(* IEC 61131-3 sources: Yaha/Documentation/Infomaterial/OSCAT/pcworx_basic_333/module_export (part 7) *)

(* ---- BIT_LOAD_DW.ST ---- *)
(*@PROPERTIES_EX@
TYPE: POU
LOCALE: 0
IEC_LANGUAGE: ST
PLC_TYPE: independent
PROC_TYPE: independent
GROUP: LOGIC.GATE_LOGIC
*)
(*@KEY@:DESCRIPTION*)
version 1.1	16. mar 2008
programmer 	hugo
tested by	tobias

this function loads a bit into a DWord at position pos.
(*@KEY@:END_DESCRIPTION*)
FUNCTION BIT_LOAD_DW:DWORD

(*Group:Default*)

VAR_INPUT
	IN :	DWORD;
	VAL :	BOOL;
	POS :	INT;
END_VAR

(*@KEY@: WORKSHEET
NAME: BIT_LOAD_DW
IEC_LANGUAGE: ST
*)
IF val THEN
	BIT_LOAD_DW := in OR SHL(DWORD#1,pos);
ELSE
	BIT_LOAD_DW := in AND (NOT SHL(DWORD#1,pos));
END_IF;

(* revision history
hm	29. feb 2008	rev 1.0
	original version

hm	16. mar 2008	rev 1.1
	change input bit to val for compatibility reasons
*)
(*@KEY@: END_WORKSHEET *)
END_FUNCTION

(* ---- BIT_LOAD_DW2.ST ---- *)
(*@PROPERTIES_EX@
TYPE: POU
LOCALE: 0
IEC_LANGUAGE: ST
PLC_TYPE: independent
PROC_TYPE: independent
GROUP: LOGIC.GATE_LOGIC
*)
(*@KEY@:DESCRIPTION*)
version 1.0 18. oct. 2008
programmer 	hugo
tested by	tobias

this function loads N bits of D at pos P in DWORD I
(*@KEY@:END_DESCRIPTION*)
FUNCTION BIT_LOAD_DW2:DWORD

(*Group:Default*)

VAR_INPUT
	I :	DWORD;
	D :	BOOL;
	P :	INT;
	N :	INT;
END_VAR

(*@KEY@: WORKSHEET
NAME: BIT_LOAD_DW2
IEC_LANGUAGE: ST
*)
IF D THEN
	BIT_LOAD_DW2 := ROL(SHR(DWORD#16#FFFFFFFF, 32 - N) OR ROR(I, P), P);
ELSE
	BIT_LOAD_DW2 := ROL(SHL(DWORD#16#FFFFFFFF, N) AND ROR(I, P), P);
END_IF;

(* revision history
hm	18. oct. 2008	rev 1.0
	original version

*)
(*@KEY@: END_WORKSHEET *)
END_FUNCTION

(* ---- BIT_LOAD_W.ST ---- *)
(*@PROPERTIES_EX@
TYPE: POU
LOCALE: 0
IEC_LANGUAGE: ST
PLC_TYPE: independent
PROC_TYPE: independent
GROUP: LOGIC.GATE_LOGIC
*)
(*@KEY@:DESCRIPTION*)
version 1.1	16. mar 2008
programmer 	hugo
tested by	tobias

this function loads a bit into a Word at position pos.
(*@KEY@:END_DESCRIPTION*)
FUNCTION BIT_LOAD_W:WORD

(*Group:Default*)

VAR_INPUT
	IN :	WORD;
	VAL :	BOOL;
	POS :	INT;
END_VAR

(*@KEY@: WORKSHEET
NAME: BIT_LOAD_W
IEC_LANGUAGE: ST
*)
IF VAL THEN
	BIT_LOAD_W := in OR SHL(WORD#1,pos);
ELSE
	BIT_LOAD_W := in AND (NOT SHL(WORD#1,pos));
END_IF;

(* revision history
hm	29. feb 2008	rev 1.0
	original version

hm	16. mar 2008	rev 1.1
	change input bit to val for compatibility reasons
*)
(*@KEY@: END_WORKSHEET *)
END_FUNCTION

(* ---- BIT_LOAD_W2.ST ---- *)
(*@PROPERTIES_EX@
TYPE: POU
LOCALE: 0
IEC_LANGUAGE: ST
PLC_TYPE: independent
PROC_TYPE: independent
GROUP: LOGIC.GATE_LOGIC
*)
(*@KEY@:DESCRIPTION*)
version 1.0 18. oct. 2008
programmer 	hugo
tested by	tobias

this function loads N bits of D at pos P in WORD I
(*@KEY@:END_DESCRIPTION*)
FUNCTION BIT_LOAD_W2:WORD

(*Group:Default*)

VAR_INPUT
	I :	WORD;
	D :	BOOL;
	P :	INT;
	N :	INT;
END_VAR

(*@KEY@: WORKSHEET
NAME: BIT_LOAD_W2
IEC_LANGUAGE: ST
*)
IF D THEN
	BIT_LOAD_W2 := ROL(SHR(WORD#16#FFFF, 16 - N) OR ROR(I, P), P);
ELSE
	BIT_LOAD_W2 := ROL(SHL(WORD#16#FFFF, N) AND ROR(I, P), P);
END_IF;

(* revision history
hm	18. oct. 2008	rev 1.0
	original version

*)
(*@KEY@: END_WORKSHEET *)
END_FUNCTION

(* ---- BIT_OF_DWORD.ST ---- *)
(*@PROPERTIES_EX@
TYPE: POU
LOCALE: 0
IEC_LANGUAGE: ST
PLC_TYPE: independent
PROC_TYPE: independent
GROUP: LOGIC.GATE_LOGIC
*)
(*@KEY@:DESCRIPTION*)
version 1.2	6. jun. 2008
programmer 	hugo
tested by	tobias

this function extracts a single bit from the nth position from right (right is lowest bit)
the lowest Bit (Bit0 from in) is selected with N=0.
(*@KEY@:END_DESCRIPTION*)
FUNCTION BIT_OF_DWORD:BOOL

(*Group:Default*)

VAR_INPUT
	IN :	DWORD;
	N :	INT;
END_VAR

(*@KEY@: WORKSHEET
NAME: BIT_OF_DWORD
IEC_LANGUAGE: ST
*)
BIT_OF_DWORD := (SHR_DWORD(in,n) AND DWORD#1) > DWORD#0;

(* old code used before rev 1.1
temp := SHR(in,n);
Bit_of_Dword := temp.0;
*)

(* revision history
hm	4. aug. 2006	rev 1.0
	original version

hm	29. feb 2008	rev 1.1
	improved performance

hm	6. jun. 2008	rev 1.2
	changes type of input N from byte to int
*)
(*@KEY@: END_WORKSHEET *)
END_FUNCTION

(* ---- BIT_TOGGLE_B.ST ---- *)
(*@PROPERTIES_EX@
TYPE: POU
LOCALE: 0
IEC_LANGUAGE: ST
PLC_TYPE: independent
PROC_TYPE: independent
GROUP: LOGIC.GATE_LOGIC
*)
(*@KEY@:DESCRIPTION*)
version 1.0 18. oct. 2008
programmer 	hugo
tested by	tobias

this function toggles a bit of a BYTE at position pos.
(*@KEY@:END_DESCRIPTION*)
FUNCTION BIT_TOGGLE_B:BYTE

(*Group:Default*)

VAR_INPUT
	IN :	BYTE;
	POS :	INT;
END_VAR

(*@KEY@: WORKSHEET
NAME: BIT_TOGGLE_B
IEC_LANGUAGE: ST
*)
BIT_TOGGLE_B := SHL(BYTE#1, POS) XOR IN;

(* revision history
hm	18. oct. 2008	rev 1.0
	original version

*)
(*@KEY@: END_WORKSHEET *)
END_FUNCTION

(* ---- BIT_TOGGLE_DW.ST ---- *)
(*@PROPERTIES_EX@
TYPE: POU
LOCALE: 0
IEC_LANGUAGE: ST
PLC_TYPE: independent
PROC_TYPE: independent
GROUP: LOGIC.GATE_LOGIC
*)
(*@KEY@:DESCRIPTION*)
version 1.0 18. oct. 2008
programmer 	hugo
tested by	tobias

this function toggles a bit of a WORD at position pos.
(*@KEY@:END_DESCRIPTION*)
FUNCTION BIT_TOGGLE_DW:DWORD

(*Group:Default*)

VAR_INPUT
	IN :	DWORD;
	POS :	INT;
END_VAR

(*@KEY@: WORKSHEET
NAME: BIT_TOGGLE_DW
IEC_LANGUAGE: ST
*)
BIT_TOGGLE_DW := SHL(DWORD#1, POS) XOR IN;

(* revision history
hm	18. oct. 2008	rev 1.0
	original version

*)
(*@KEY@: END_WORKSHEET *)
END_FUNCTION

(* ---- BIT_TOGGLE_W.ST ---- *)
(*@PROPERTIES_EX@
TYPE: POU
LOCALE: 0
IEC_LANGUAGE: ST
PLC_TYPE: independent
PROC_TYPE: independent
GROUP: LOGIC.GATE_LOGIC
*)
(*@KEY@:DESCRIPTION*)
version 1.0 18. oct. 2008
programmer 	hugo
tested by	tobias

this function toggles a bit of a WORD at position pos.
(*@KEY@:END_DESCRIPTION*)
FUNCTION BIT_TOGGLE_W:WORD

(*Group:Default*)

VAR_INPUT
	IN :	WORD;
	POS :	INT;
END_VAR

(*@KEY@: WORKSHEET
NAME: BIT_TOGGLE_W
IEC_LANGUAGE: ST
*)
BIT_TOGGLE_W := SHL(WORD#1, POS) XOR IN;

(* revision history
hm	18. oct. 2008	rev 1.0
	original version

*)
(*@KEY@: END_WORKSHEET *)
END_FUNCTION

(* ---- BYTE_OF_BIT.ST ---- *)
(*@PROPERTIES_EX@
TYPE: POU
LOCALE: 0
IEC_LANGUAGE: ST
PLC_TYPE: independent
PROC_TYPE: independent
GROUP: LOGIC.GATE_LOGIC
*)
(*@KEY@:DESCRIPTION*)
version 1.1	 18. feb 2006
programmer 	hugo
tested by	tobias

this function creates a byte from 8 individual bits
(*@KEY@:END_DESCRIPTION*)
FUNCTION BYTE_OF_BIT:BYTE

(*Group:Default*)

VAR_INPUT
	B0 :	BOOL;
	B1 :	BOOL;
	B2 :	BOOL;
	B3 :	BOOL;
	B4 :	BOOL;
	B5 :	BOOL;
	B6 :	BOOL;
	B7 :	BOOL;
END_VAR

(*@KEY@: WORKSHEET
NAME: BYTE_OF_BIT
IEC_LANGUAGE: ST
*)
Byte_of_bit := SHL_BYTE(SHL_BYTE(SHL_BYTE(SHL_BYTE(SHL_BYTE(SHL_BYTE(SHL_BYTE(BOOL_TO_BYTE(B7),1) OR BOOL_TO_BYTE(B6),1)
 OR BOOL_TO_BYTE(B5),1) OR BOOL_TO_BYTE(B4),1) OR BOOL_TO_BYTE(B3),1) OR BOOL_TO_BYTE(B2),1)
 OR BOOL_TO_BYTE(B1),1) OR BOOL_TO_BYTE(B0);

(* revision history

hm	4. aug 2006		rev 1.0
	original version

hm	18. feb. 2008	rev 1.1
	improved performance

*)
(*@KEY@: END_WORKSHEET *)
END_FUNCTION

(* ---- BYTE_OF_DWORD.ST ---- *)
(*@PROPERTIES_EX@
TYPE: POU
LOCALE: 0
IEC_LANGUAGE: ST
PLC_TYPE: independent
PROC_TYPE: independent
GROUP: LOGIC.GATE_LOGIC
*)
(*@KEY@:DESCRIPTION*)
version 1.2	30. oct. 2008
programmer 	hugo
tested by	oscat

this function extracts a single byte from the nth position from right (right is lowest byte)
the lower byte (starting with Bit0 from in) is selected with N=0.
(*@KEY@:END_DESCRIPTION*)
FUNCTION BYTE_OF_DWORD:BYTE

(*Group:Default*)

VAR_INPUT
	IN :	DWORD;
	N :	BYTE;
END_VAR

(*@KEY@: WORKSHEET
NAME: BYTE_OF_DWORD
IEC_LANGUAGE: ST
*)
BYTE_OF_DWORD := DWORD_TO_BYTE(SHR(in,_BYTE_TO_INT(SHL(n,3))));

(* revision history
hm	17. jan 2007	rev 1.0
	original version

hm	2. jan 2008		rev 1.1
	improved performance

hm	30. oct. 2008	rev 1.2
	improved performance
*)
(*@KEY@: END_WORKSHEET *)
END_FUNCTION

(* ---- BYTE_TO_GRAY.ST ---- *)
(*@PROPERTIES_EX@
TYPE: POU
LOCALE: 0
IEC_LANGUAGE: ST
PLC_TYPE: independent
PROC_TYPE: independent
GROUP: LOGIC.GATE_LOGIC
*)
(*@KEY@:DESCRIPTION*)
version 1.0	9. nov. 2009
programmer 	hugo
tested by	oscat

this function converts a binary to gray code
(*@KEY@:END_DESCRIPTION*)
FUNCTION BYTE_TO_GRAY:BYTE

(*Group:Default*)

VAR_INPUT
	IN :	BYTE;
END_VAR

(*@KEY@: WORKSHEET
NAME: BYTE_TO_GRAY
IEC_LANGUAGE: ST
*)
BYTE_TO_GRAY := IN XOR SHR(IN,1);

(* revision history
hm	9. nov. 2009	rev 1.0
	original version

*)

(*@KEY@: END_WORKSHEET *)
END_FUNCTION

(* ---- BYTE_TO_RANGE.ST ---- *)
(*@PROPERTIES_EX@
TYPE: POU
LOCALE: 0
IEC_LANGUAGE: ST
PLC_TYPE: independent
PROC_TYPE: independent
GROUP: ENGINEERING.SIGNAL_PROCESSING
*)
(*@KEY@:DESCRIPTION*)
version 1.0	9. jan 2008
programmer 	hugo
tested by	tobias

Byte_to_Range converts a Byte into a real between low and high.
(*@KEY@:END_DESCRIPTION*)
FUNCTION BYTE_TO_RANGE:REAL

(*Group:Default*)

VAR_INPUT
	X :	BYTE;
	LOW :	REAL;
	HIGH :	REAL;
END_VAR

(*@KEY@: WORKSHEET
NAME: BYTE_TO_RANGE
IEC_LANGUAGE: ST
*)
Byte_to_Range := (high - low) * _BYTE_TO_REAL(X) / 255.0 + low;

(* revision history
hm	9. jan 2008		rev 1.0
	original version

*)
(*@KEY@: END_WORKSHEET *)
END_FUNCTION

(* ---- C_TO_F.ST ---- *)
(*@PROPERTIES_EX@
TYPE: POU
LOCALE: 0
IEC_LANGUAGE: ST
PLC_TYPE: independent
PROC_TYPE: independent
GROUP: ENGINEERING.CONVERSION
*)
(*@KEY@:DESCRIPTION*)
version 1.1	11. mar. 2009
programmer 	hugo
tested by	tobias

this function converts celsius  to fahrenheit
(*@KEY@:END_DESCRIPTION*)
FUNCTION C_TO_F:REAL

(*Group:Default*)

VAR_INPUT
	CELSIUS :	REAL;
END_VAR

(*@KEY@: WORKSHEET
NAME: C_TO_F
IEC_LANGUAGE: ST
*)
C_TO_F := celsius * 1.8 + 32.0;

(* revision history

hm	4. aug. 2006	rev 1.0
	original version

hm	11. mar. 2009	rev 1.1
	real constants updated to new systax using dot

*)
(*@KEY@: END_WORKSHEET *)
END_FUNCTION

(* ---- C_TO_K.ST ---- *)
(*@PROPERTIES_EX@
TYPE: POU
LOCALE: 0
IEC_LANGUAGE: ST
PLC_TYPE: independent
PROC_TYPE: independent
GROUP: ENGINEERING.CONVERSION
*)
(*@KEY@:DESCRIPTION*)
version 1.1	19. aug 2009
programmer 	hugo
tested by		tobias

this function converts celsius to kelvin
(*@KEY@:END_DESCRIPTION*)
FUNCTION C_TO_K:REAL

(*Group:Default*)

VAR_INPUT
	CELSIUS :	REAL;
END_VAR

(*@KEY@: WORKSHEET
NAME: C_TO_K
IEC_LANGUAGE: ST
*)
C_to_K := Celsius - 273.15;

(* revision history

hm	4. aug 2006	rev 1.0
	original version

hm	19. aug 2009	rev 1.1
	fixed calculation error

*)

(*@KEY@: END_WORKSHEET *)
END_FUNCTION

(* ---- CAUCHY.ST ---- *)
(*@PROPERTIES_EX@
TYPE: POU
LOCALE: 0
IEC_LANGUAGE: ST
PLC_TYPE: independent
PROC_TYPE: independent
GROUP: MATHEMATICAL.MATHE
*)
(*@KEY@:DESCRIPTION*)
version 1.0	26. oct. 2008
programmer 	hugo
tested by	tobias

this function calculates the Cauchy distribution function
(*@KEY@:END_DESCRIPTION*)
FUNCTION CAUCHY:REAL

(*Group:Default*)

VAR_INPUT
	X :	REAL;
	T :	REAL;
	U :	REAL;
END_VAR

VAR
	tmp :	REAL;
END_VAR

(*@KEY@: WORKSHEET
NAME: CAUCHY
IEC_LANGUAGE: ST
*)
tmp := x - t;
CAUCHY := 0.318309886183791 * U / (U*U + tmp*tmp);

(* revision hisdtory
hm	26. oct. 2008	rev 1.0
	original version

*)
(*@KEY@: END_WORKSHEET *)
END_FUNCTION

(* ---- CAUCHYCD.ST ---- *)
(*@PROPERTIES_EX@
TYPE: POU
LOCALE: 0
IEC_LANGUAGE: ST
PLC_TYPE: independent
PROC_TYPE: independent
GROUP: MATHEMATICAL.MATHE
*)
(*@KEY@:DESCRIPTION*)
version 1.0	26. oct. 2008
programmer 	hugo
tested by	tobias

this function calculates the Cauchy distribution function
(*@KEY@:END_DESCRIPTION*)
FUNCTION CAUCHYCD:REAL

(*Group:Default*)

VAR_INPUT
	X :	REAL;
	T :	REAL;
	U :	REAL;
END_VAR

(*@KEY@: WORKSHEET
NAME: CAUCHYCD
IEC_LANGUAGE: ST
*)
CAUCHYCD := 0.5 + 0.318309886183791 * ATAN((X - T) / U);

(* revision hisdtory
hm	26. oct. 2008	rev 1.0
	original version

*)
(*@KEY@: END_WORKSHEET *)
END_FUNCTION

(* ---- CEIL.ST ---- *)
(*@PROPERTIES_EX@
TYPE: POU
LOCALE: 0
IEC_LANGUAGE: ST
PLC_TYPE: independent
PROC_TYPE: independent
GROUP: MATHEMATICAL.MATHE
*)
(*@KEY@:DESCRIPTION*)
version 1.0	7 feb 2007
programmer 	hugo
tested by	tobias

This is a rounding function which returns the smallest possible integer which is greater or equal to X.
ceil(3.14) = 4
ceil(-3.14) = -3
(*@KEY@:END_DESCRIPTION*)
FUNCTION CEIL:INT

(*Group:Default*)

VAR_INPUT
	X :	REAL;
END_VAR

(*@KEY@: WORKSHEET
NAME: CEIL
IEC_LANGUAGE: ST
*)
CEIL := REAL_TO_INT(x);
IF INT_TO_REAL(CEIL) < X THEN
        CEIL := CEIL + 1;
END_IF;

(* code before rev 1.1
CEIL := D_TRUNC(X);
IF CEIL < X THEN
	ceil := ceil + 1;
END_IF;
*)

(* revision history
hm		7. feb. 2007	rev 1.0
	original version

hm		21. mar. 2008	rev 1.1
	use REAL_TO_INT instead of trunc for compatibility reasons

*)
(*@KEY@: END_WORKSHEET *)
END_FUNCTION

(* ---- CEIL2.ST ---- *)
(*@PROPERTIES_EX@
TYPE: POU
LOCALE: 0
IEC_LANGUAGE: ST
PLC_TYPE: independent
PROC_TYPE: independent
GROUP: MATHEMATICAL.MATHE
*)
(*@KEY@:DESCRIPTION*)
version 1.3	10. mar. 2009
programmer 	hugo
tested by	tobias

This is a rounding function which returns the smallest possible integer which is greater or equal to X.
ceil2(3.14) = 4
ceil2(-3.14) = -3

(*@KEY@:END_DESCRIPTION*)
FUNCTION CEIL2:DINT

(*Group:Default*)

VAR_INPUT
	X :	REAL;
END_VAR

(*@KEY@: WORKSHEET
NAME: CEIL2
IEC_LANGUAGE: ST
*)
CEIL2 := _REAL_TO_DINT(x);
IF DINT_TO_REAL(CEIL2) < X THEN
        CEIL2 := CEIL2 + DINT#1;
END_IF;

(* revision history
hm	21. mar. 2008	rev 1.0
	original version

hm	4. apr. 2008	rev 1.1
	added type conversion to avoid warnings under codesys 3.0

hm	30. jun. 2008	rev 1.2
	added type conversion to avoid warnings under codesys 3.0

hm	10. mar. 2009	rev 1.3
	use correct statement real_to_DINT

*)
(*@KEY@: END_WORKSHEET *)
END_FUNCTION

(* ---- CHECK_PARITY.ST ---- *)
(*@PROPERTIES_EX@
TYPE: POU
LOCALE: 0
IEC_LANGUAGE: ST
PLC_TYPE: independent
PROC_TYPE: independent
GROUP: LOGIC.GATE_LOGIC
*)
(*@KEY@:DESCRIPTION*)
version 1.3	18 feb 2008
programmer 	hugo
tested by	tobias

this function checks for an even partity for a dword and partity bit.
(*@KEY@:END_DESCRIPTION*)
FUNCTION CHECK_PARITY:BOOL

(*Group:Default*)

VAR_INPUT
	IN :	DWORD;
	P :	BOOL;
END_VAR

VAR
	in2 :	DWORD;
END_VAR

(*@KEY@: WORKSHEET
NAME: CHECK_PARITY
IEC_LANGUAGE: ST
*)
in2:=in;
check_parity := NOT p;
WHILE in2 > DWORD#0 DO
	check_parity := check_parity XOR BIT_OF_DWORD(in2,0) XOR BIT_OF_DWORD(in2,1) XOR BIT_OF_DWORD(in2,2) XOR BIT_OF_DWORD(in2,3);
	in2 := SHR(in2,4);
END_WHILE;

(* code before rev 1.2
WHILE in > 0 DO
	IF in.0 THEN cnt := cnt + 1; END_IF;
	in := SHR(in,1);
END_WHILE;
check_parity := even(cnt) XOR P;
*)

(* revision history

rev 1.0 HM  1.oct.2006

rev 1.1 hm	10.sep.2007
	changed algorithm to improove performance

rev 1.2	hm	8 dec 2007
	changed algorithm to improove performance

rev 1.3 hm	18. feb 2008
	changed algorithm to improove performance
*)
(*@KEY@: END_WORKSHEET *)
END_FUNCTION

(* ---- CIRCLE_A.ST ---- *)
(*@PROPERTIES_EX@
TYPE: POU
LOCALE: 0
IEC_LANGUAGE: ST
PLC_TYPE: independent
PROC_TYPE: independent
GROUP: MATHEMATICAL.GEOMETRY
*)
(*@KEY@:DESCRIPTION*)
version 1.2	22. feb 2008
programmer 	hugo
tested by	tobias

circle_A calculates the Area of a circle segement if ax = 360 the whole circle is calculated
(*@KEY@:END_DESCRIPTION*)
FUNCTION CIRCLE_A:REAL

(*Group:Default*)

VAR_INPUT
	RX :	REAL;
	AX :	REAL;
END_VAR

(*@KEY@: WORKSHEET
NAME: CIRCLE_A
IEC_LANGUAGE: ST
*)
circle_A := Rx * RX * 8.726646E-3 * Ax;

(* revision histroy
hm	16. oct 2007	rev 1.0
	original version

hm	4. dec 2007		rev 1.1
	changed code for better performance

hm	22. feb 2008	rev 1.2
	improved performance
*)
(*@KEY@: END_WORKSHEET *)
END_FUNCTION

(* ---- CIRCLE_C.ST ---- *)
(*@PROPERTIES_EX@
TYPE: POU
LOCALE: 0
IEC_LANGUAGE: ST
PLC_TYPE: independent
PROC_TYPE: independent
GROUP: MATHEMATICAL.GEOMETRY
*)
(*@KEY@:DESCRIPTION*)
version 1.1	22 feb 2008
programmer 	hugo
tested by	tobias

circle_C calculates the Circumference of a circle  if ax = 360 the whole circle is calculated
(*@KEY@:END_DESCRIPTION*)
FUNCTION CIRCLE_C:REAL

(*Group:Default*)

VAR_INPUT
	RX :	REAL;
	AX :	REAL;
END_VAR

(*@KEY@: WORKSHEET
NAME: CIRCLE_C
IEC_LANGUAGE: ST
*)
circle_C := 1.7453293E-2 * Rx * Ax;

(* revision histroy
hm	16. oct 2007	rev 1.0
	original version

hm	22. feb 2008	rev 1.1
	improved performance
*)
(*@KEY@: END_WORKSHEET *)
END_FUNCTION

(* ---- CIRCLE_SEG.ST ---- *)
(*@PROPERTIES_EX@
TYPE: POU
LOCALE: 0
IEC_LANGUAGE: ST
PLC_TYPE: independent
PROC_TYPE: independent
GROUP: MATHEMATICAL.GEOMETRY
*)
(*@KEY@:DESCRIPTION*)
version 1.0	10. Mar 2010
programmer 	hugo
tested by	tobias

CIRCLE_SEG calculates the Area of a circle segement enclosed between a sectant line and the circumference.

(*@KEY@:END_DESCRIPTION*)
FUNCTION CIRCLE_SEG:REAL

(*Group:Default*)

VAR_INPUT
	RX :	REAL;
	HX :	REAL;
END_VAR

(*@KEY@: WORKSHEET
NAME: CIRCLE_SEG
IEC_LANGUAGE: ST
*)
IF RX > 0.0 THEN
	CIRCLE_SEG := 2.0 * ACOS(1.0 - LIMIT(0.0, HX / RX, 2.0));
	CIRCLE_SEG := (CIRCLE_SEG - SIN(CIRCLE_SEG)) * RX * RX * 0.5;
END_IF;

(* revision histroy
hm	10. mar 2010	rev 1.0
	original version

*)
(*@KEY@: END_WORKSHEET *)
END_FUNCTION

(* ---- CMP.ST ---- *)
(*@PROPERTIES_EX@
TYPE: POU
LOCALE: 0
IEC_LANGUAGE: ST
PLC_TYPE: independent
PROC_TYPE: independent
GROUP: MATHEMATICAL.MATHE
*)
(*@KEY@:DESCRIPTION*)
version 1.1	10. mar. 2009
programmer 	hugo
tested by	tobias

this function checks two inputs x and y if they are identical with the first N digits
example : cmp(3.141516,3.141517,6 is true.

(*@KEY@:END_DESCRIPTION*)
FUNCTION CMP:BOOL

(*Group:Default*)

VAR_INPUT
	X :	REAL;
	Y :	REAL;
	N :	INT;
END_VAR

VAR
	tmp :	REAL;
END_VAR

(*@KEY@: WORKSHEET
NAME: CMP
IEC_LANGUAGE: ST
*)
tmp := ABS(x);
IF tmp > 0.0 THEN
	tmp := EXP10(INT_TO_REAL(FLOOR(LOG(tmp))-N+1));
ELSE
	tmp := EXP10(tmp);
END_IF;
CMP := ABS(X - Y) < tmp;

(* revision history
hm	12. mar. 2008	rev 1.0
	original version

hm	10. mar. 2009	rev 1.1
	added type conversion for compatibility reasons
*)

(*@KEY@: END_WORKSHEET *)
END_FUNCTION

(* ---- CONE_V.ST ---- *)
(*@PROPERTIES_EX@
TYPE: POU
LOCALE: 0
IEC_LANGUAGE: ST
PLC_TYPE: independent
PROC_TYPE: independent
GROUP: MATHEMATICAL.GEOMETRY
*)
(*@KEY@:DESCRIPTION*)
version 1.1	4 dec 2007
programmer 	hugo
tested by	tobias

cone_V calculates the Volume of a cone
(*@KEY@:END_DESCRIPTION*)
FUNCTION CONE_V:REAL

(*Group:Default*)

VAR_INPUT
	RX :	REAL;
	HX :	REAL;
END_VAR

(*@KEY@: WORKSHEET
NAME: CONE_V
IEC_LANGUAGE: ST
*)
cone_V := 1.047197551 * RX * RX * hx;

(* revision histroy
hm	17. oct 2007	rev 1.0
	original version

hm	4. dec 2007		rev 1.1
	changed code for better performance

hm	22. feb 2008	rev 1.2
	changed code for better performance
*)
(*@KEY@: END_WORKSHEET *)
END_FUNCTION

(* ---- COSH.ST ---- *)
(*@PROPERTIES_EX@
TYPE: POU
LOCALE: 0
IEC_LANGUAGE: ST
PLC_TYPE: independent
PROC_TYPE: independent
GROUP: MATHEMATICAL.MATHE
*)
(*@KEY@:DESCRIPTION*)
version 1.3	10. mar. 2009
programmer 	hugo
tested by	tobias

this function calculates the cos hyperbolicus

(*@KEY@:END_DESCRIPTION*)
FUNCTION COSH:REAL

(*Group:Default*)

VAR_INPUT
	X :	REAL;
END_VAR

VAR
	t :	REAL;
END_VAR

(*@KEY@: WORKSHEET
NAME: COSH
IEC_LANGUAGE: ST
*)
T := EXP(X);
COSH := (1.0 / T + T) * 0.5;

(* revision histroy
hm	12.1.2007	rev 1.0
	original version

hm	1.12.2007	rev 1.1
	changed code to improve performance

hm	5. jan 2008	rev 1.2
	further performance improvement

hm	10. mar. 2009	rev 1.3
	real constants updated to new systax using dot
*)
(*@KEY@: END_WORKSHEET *)
END_FUNCTION

(* ---- COTH.ST ---- *)
(*@PROPERTIES_EX@
TYPE: POU
LOCALE: 0
IEC_LANGUAGE: ST
PLC_TYPE: independent
PROC_TYPE: independent
GROUP: MATHEMATICAL.MATHE
*)
(*@KEY@:DESCRIPTION*)
version 1.4	10. mar. 2009
programmer 	hugo
tested by	tobias

this function calculates the cotangens hyperbolicus
(*@KEY@:END_DESCRIPTION*)
FUNCTION COTH:REAL

(*Group:Default*)

VAR_INPUT
	X :	REAL;
END_VAR

(*@KEY@: WORKSHEET
NAME: COTH
IEC_LANGUAGE: ST
*)
IF X > 20.0 THEN
	COTH :=1.0;
ELSIF X < -20.0 THEN
	COTH := -1.0;
ELSE
	COTH := 1.0 + 2.0 / (EXP(X * 2.0) - 1.0);
END_IF;

(* revision histroy
hm		12.1.2007	rev 1.0
	original version

hm	1.12.2007		rev 1.1
	changed code to improve performance

hm	8. jan 2008	rev 1.2
	further improvement in performance

hm	10. mar 2008	rev 1.3
	extended range of valid inputs to +/- INV
	changed formula for better accuracy

hm	10. mar. 2009	rev 1.4
	real constants updated to new systax using dot
*)
(*@KEY@: END_WORKSHEET *)
END_FUNCTION

(* ---- CTRL_IN.ST ---- *)
(*@PROPERTIES_EX@
TYPE: POU
LOCALE: 0
IEC_LANGUAGE: ST
PLC_TYPE: independent
PROC_TYPE: independent
GROUP: ENGINEERING.CONTROL
*)
(*@KEY@:DESCRIPTION*)
version 1.0	2. jun 2008
programmer 	hugo
tested by	tobias
(*@KEY@:END_DESCRIPTION*)
FUNCTION CTRL_IN:REAL

(*Group:Default*)

VAR_INPUT
	SET_POINT :	REAL;
	ACTUAL :	REAL;
	NOISE :	REAL;
END_VAR

(*@KEY@: WORKSHEET
NAME: CTRL_IN
IEC_LANGUAGE: ST
*)
(* calculate the process error DIFF *)
CTRL_IN := DEAD_ZONE(SET_POINT - ACTUAL, NOISE);

(* revision history
hm 	2. jun. 2008 	rev 1.0
	original version

*)
(*@KEY@: END_WORKSHEET *)
END_FUNCTION

(* ---- D_TRUNC.ST ---- *)
(*@PROPERTIES_EX@
TYPE: POU
LOCALE: 0
IEC_LANGUAGE: ST
PLC_TYPE: independent
PROC_TYPE: independent
GROUP: MATHEMATICAL.MATHE
*)
(*@KEY@:DESCRIPTION*)
version 1.2	10. mar. 2009
programmer 	hugo
tested by	oscat

d_trunc truncates a real to a dint 1.5 will be 1 and -1.5 will be -1
d_trunc is necessary because many systems do not offer a trunc to a dint
also real_to_dint will not deliver the same result on different systems

(*@KEY@:END_DESCRIPTION*)
FUNCTION D_TRUNC:DINT

(*Group:Default*)

VAR_INPUT
	X :	REAL;
END_VAR

(*@KEY@: WORKSHEET
NAME: D_TRUNC
IEC_LANGUAGE: ST
*)
D_TRUNC := TRUNC_DINT(X);

(*
D_TRUNC := REAL_TO_DINT(X);
IF X > 0.0 THEN
	IF DINT_TO_REAL(D_TRUNC) > X THEN D_TRUNC := D_TRUNC - DINT#1; END_IF;
ELSE
	IF DINT_TO_REAL(D_TRUNC) < X THEN D_TRUNC := D_TRUNC + DINT#1; END_IF;
END_IF;
*)

(* for systems that support a dint truncation this routine can be replaced by trunc() *)

(* revision history
hm	21. mar. 2008	rev 1.0
	original version

hm	31. oct. 2008	rev 1.1
	optimized performance

hm	10. mar. 2009	rev 1.2
	real constants updated to new systax using dot
*)
(*@KEY@: END_WORKSHEET *)
END_FUNCTION

(* ---- DATE_ADD.ST ---- *)
(*@PROPERTIES_EX@
TYPE: POU
LOCALE: 0
IEC_LANGUAGE: ST
PLC_TYPE: independent
PROC_TYPE: independent
GROUP: TIME_DATE
*)
(*@KEY@:DESCRIPTION*)
version 1.8		22. mar. 2011
programmer 	    hugo
tested by		oscat

date_add adds days, weeks, month or years to a date.
negative inputs are allowed for subtraction.

(*@KEY@:END_DESCRIPTION*)
FUNCTION DATE_ADD:UDINT

(*Group:Default*)

VAR_INPUT
	IDATE :	UDINT;
	D :	INT;
	W :	INT;
	M :	INT;
	Y :	INT;
END_VAR

VAR
	mo :	INT;
	yr :	INT;
	dm :	INT;
END_VAR

(*@KEY@: WORKSHEET
NAME: DATE_ADD
IEC_LANGUAGE: ST
*)
DATE_ADD := IDATE + INT_TO_UDINT(D + W * 7) * UDINT#86400;
yr := Y + YEAR_OF_DATE(DATE_ADD);
mo := M + MONTH_OF_DATE(DATE_ADD);
dm := DAY_OF_MONTH(DATE_ADD);
WHILE mo > 12 DO
	mo := mo - 12;
	yr := yr + 1;
END_WHILE;
WHILE mo < 1 DO
	mo := mo + 12;
	yr := yr - 1;
END_WHILE;
DATE_ADD := SET_DATE(yr, mo, dm);

(* revision history

hm 27.12.2006	rev 1.0
	nrw module

hm 12.4.2007		rev 1.1
	corrected an error while date would be incorrect when year  = 0

hm	1.11.2007		rev 1.2
	added int_to_dword stetements to avoid possible overrun with möller ecp4

hm	22. mar. 2008	rev 1.3
	fixed some bugs when month was negative

hm	7. oct. 2008	rev 1.4
	changed function year to year_of_date
	changed function month to month_of_date

hm	29. mar. 2009	rev 1.5
	improved performance

hm	27. jan. 2011	rev 1.6
	faster code

hm	2. feb. 2011		rev 1.7
	fixed an error, weeks not calculated

hm	22. mar. 2011	rev 1.8
	fixed an error in formula
*)
(*@KEY@: END_WORKSHEET *)
END_FUNCTION

(* ---- DAY_OF_DATE.ST ---- *)
(*@PROPERTIES_EX@
TYPE: POU
LOCALE: 0
IEC_LANGUAGE: ST
PLC_TYPE: independent
PROC_TYPE: independent
GROUP: TIME_DATE
*)
(*@KEY@:DESCRIPTION*)
version 1.1	9. oct. 2008
programmer 	hugo
tested by	oscat

TIMER_P4 is a programmable universal timer.
(*@KEY@:END_DESCRIPTION*)
FUNCTION DAY_OF_DATE:DINT

(*Group:Default*)

VAR_INPUT
	IDATE :	UDINT;
END_VAR

(*@KEY@: WORKSHEET
NAME: DAY_OF_DATE
IEC_LANGUAGE: ST
*)
day_of_date := UDINT_TO_DINT(idate / UDINT#86400);

(* revision history
hm		16.9.2007		rev 1.0
	original version

hm		1. okt 2007		rev 1.1
	added step7 compatibility

hm		22. mar. 2008	rev 1.2
	changed output from int to Dint because the total date range is 49710 days

hm		7. apr. 2008	rev 1.3
	deleted unused step7 code

*)
(*@KEY@: END_WORKSHEET *)
END_FUNCTION

(* ---- DAY_OF_MONTH.ST ---- *)
(*@PROPERTIES_EX@
TYPE: POU
LOCALE: 0
IEC_LANGUAGE: ST
PLC_TYPE: independent
PROC_TYPE: independent
GROUP: TIME_DATE
*)
(*@KEY@:DESCRIPTION*)
version 2.1	10. mar. 2009
programmer 	hugo
tested by	tobias

returns the day OF month for any DATE
(*@KEY@:END_DESCRIPTION*)
FUNCTION DAY_OF_MONTH:INT

(*Group:Default*)

VAR_INPUT
	IDATE :	UDINT;
END_VAR

(*@KEY@: WORKSHEET
NAME: DAY_OF_MONTH
IEC_LANGUAGE: ST
*)
day_of_month := day_of_year(idate);

IF leap_of_Date(idate) THEN
	CASE day_of_month OF
		32..60	:	day_of_month := day_of_month - 31;
		61..91	:	day_of_month := day_of_month - 60;
		92..121 :	day_of_month := day_of_month - 91;
		122..152:	day_of_month := day_of_month - 121;
		153..182:	day_of_month := day_of_month - 152;
		183..213:	day_of_month := day_of_month - 182;
		214..244:	day_of_month := day_of_month - 213;
		245..274:	day_of_month := day_of_month - 244;
		275..305:	day_of_month := day_of_month - 274;
		306..335:	day_of_month := day_of_month - 305;
		336..366:	day_of_month := day_of_month - 335;
	END_CASE;
ELSE
	CASE day_of_month OF
		32..59	:	day_of_month := day_of_month - 31;
		60..90	:	day_of_month := day_of_month - 59;
		91..120 :	day_of_month := day_of_month - 90;
		121..151:	day_of_month := day_of_month - 120;
		152..181:	day_of_month := day_of_month - 151;
		182..212:	day_of_month := day_of_month - 181;
		213..243:	day_of_month := day_of_month - 212;
		244..273:	day_of_month := day_of_month - 243;
		274..304:	day_of_month := day_of_month - 273;
		305..334:	day_of_month := day_of_month - 304;
		335..365:	day_of_month := day_of_month - 334;
	END_CASE;
END_IF;

(*
Revision history

hm 22.1.2007		rev 1.1
	deleted unused variable day_in_year and day_in_year_begin

hm	1. okt 2007	rev 1.2
	changed code to use day_of_year and leap_of_date
	added compatibility to STEP7

hm	8. oct 2007	rev 1.3
	deleted unused variable yr

hm	8. jan 2008	rev 1.4
	improved performance

hm	25. oct. 2008	rev 2.0
	new code using setup constants

hm	10. mar. 2009	rev 2.1
	removed nested comments
*)
(*@KEY@: END_WORKSHEET *)
END_FUNCTION

(* ---- DAY_OF_WEEK.ST ---- *)
(*@PROPERTIES_EX@
TYPE: POU
LOCALE: 0
IEC_LANGUAGE: ST
PLC_TYPE: independent
PROC_TYPE: independent
GROUP: TIME_DATE
*)
(*@KEY@:DESCRIPTION*)
version 1.4	7. oct. 2008
programmer 	hugo
tested by	tobias

calculates the weekday of a week according to ISO8601
monday = 1 ..... sunday = 7
(*@KEY@:END_DESCRIPTION*)
FUNCTION DAY_OF_WEEK:INT

(*Group:Default*)

VAR_INPUT
	IDATE :	UDINT;
END_VAR

(*@KEY@: WORKSHEET
NAME: DAY_OF_WEEK
IEC_LANGUAGE: ST
*)
DAY_OF_WEEK := UDINT_TO_INT((idate / UDINT#86400 + UDINT#3) MOD UDINT#7) + INT#01;

(* revision history
hm 	21.8.06 		rev 1.1
	corrected a miscalculation

hm	23.12.2007		rev 1.2
	correction for step7

hm	7. apr. 2008	rev 1.3
	deleted unused step7 code

hm	7. oct. 2008	rev 1.4
	changed name of function from weekday to day_of_week

*)
(*@KEY@: END_WORKSHEET *)
END_FUNCTION

(* ---- DAY_OF_YEAR.ST ---- *)
(*@PROPERTIES_EX@
TYPE: POU
LOCALE: 0
IEC_LANGUAGE: ST
PLC_TYPE: independent
PROC_TYPE: independent
GROUP: TIME_DATE
*)
(*@KEY@:DESCRIPTION*)
version 1.4		28. jan. 2011
programmer 		hugo
tested by		oscat

calculates the day of the year

(*@KEY@:END_DESCRIPTION*)
FUNCTION DAY_OF_YEAR:INT

(*Group:Default*)

VAR_INPUT
	IDATE :	UDINT;
END_VAR

(*@KEY@: WORKSHEET
NAME: DAY_OF_YEAR
IEC_LANGUAGE: ST
*)
DAY_OF_YEAR := UDINT_TO_INT((DATE_TO_UDINT(idate) / UDINT#86400) MOD UDINT#1461);
IF DAY_OF_YEAR > 729 THEN
	IF DAY_OF_YEAR > 1095 THEN DAY_OF_YEAR := DAY_OF_YEAR - 1095; ELSE DAY_OF_YEAR := DAY_OF_YEAR - 729; END_IF;
ELSIF DAY_OF_YEAR > 364 THEN
	DAY_OF_YEAR := DAY_OF_YEAR - 364;
ELSE
	DAY_OF_YEAR := DAY_OF_YEAR + 1;
END_IF;

(*
DAY_OF_YEAR := DWORD_TO_INT((DATE_TO_DWORD(idate) - DATE_TO_DWORD(YEAR_BEGIN(YEAR_OF_DATE(idate)))) / 86400) + 1;
*)

(* revivision history
hm	4. aug. 2007		rev 1.0
	original version

hm	1. oct. 2007		rev 1.1
	added compatibility to STEP7

hm	4. jan. 2008		rev 1.2
	changed code for better performance

hm	7. oct. 2008		rev 1.3
	changed name of function year to year_of_date

hm	28. jan. 2011	rev 1.4
	improved code
*)
(*@KEY@: END_WORKSHEET *)
END_FUNCTION

(* ---- DAY_TO_TIME.ST ---- *)
(*@PROPERTIES_EX@
TYPE: POU
LOCALE: 0
IEC_LANGUAGE: ST
PLC_TYPE: independent
PROC_TYPE: independent
GROUP: TIME_DATE
*)
(*@KEY@:DESCRIPTION*)
version 1.1	24. feb. 2009
programmer 	hugo
tested by	tobias

converts an amount of days in real to time
(*@KEY@:END_DESCRIPTION*)
FUNCTION DAY_TO_TIME:TIME

(*Group:Default*)

VAR_INPUT
	IN :	REAL;
END_VAR

(*@KEY@: WORKSHEET
NAME: DAY_TO_TIME
IEC_LANGUAGE: ST
*)
day_to_time := DINT_TO_TIME(UDINT_TO_DINT(_REAL_TO_UDINT(IN * REAL#86400000.00)));

(* revision history
hm	4. aug. 2006	rev 1.0
	original release

hm	24. feb. 2009	rev 1.1
	renamed input to IN
*)
(*@KEY@: END_WORKSHEET *)
END_FUNCTION

(* ---- DAYS_DELTA.ST ---- *)
(*@PROPERTIES_EX@
TYPE: POU
LOCALE: 0
IEC_LANGUAGE: ST
PLC_TYPE: independent
PROC_TYPE: independent
GROUP: TIME_DATE
*)
(*@KEY@:DESCRIPTION*)
version 1.3		25. jan. 2011
programmer 		hugo
tested by		tobias

days_delta calculates the days between two dates. the days are calculated date_2 - date_1.

(*@KEY@:END_DESCRIPTION*)
FUNCTION DAYS_DELTA:DINT

(*Group:Default*)

VAR_INPUT
	DATE_1 :	UDINT;
	DATE_2 :	UDINT;
END_VAR

(*@KEY@: WORKSHEET
NAME: DAYS_DELTA
IEC_LANGUAGE: ST
*)
IF DATE_1 > DATE_2 THEN
	DAYS_DELTA := - UDINT_TO_DINT((date_1 - date_2) / UDINT#86400);
ELSE
	DAYS_DELTA :=   UDINT_TO_DINT((date_2 - date_1) / UDINT#86400);
END_IF;

(* revision history
hm	27. dec 2006	rev 1.0
	original version

hm	16.9.2007		rev 1.1
	coorected an error in formula and changed algorithm to show positive and negative delta

hm	22. mar. 2008	rev 1.2
	changed output from int to dint because the total date range is 49710 days

hm	25. jan. 2011	rev 1.3
	improved performance
*)
(*@KEY@: END_WORKSHEET *)
END_FUNCTION

(* ---- DAYS_IN_MONTH.ST ---- *)
(*@PROPERTIES_EX@
TYPE: POU
LOCALE: 0
IEC_LANGUAGE: ST
PLC_TYPE: independent
PROC_TYPE: independent
GROUP: TIME_DATE
*)
(*@KEY@:DESCRIPTION*)
version 1.0	27. mar. 2009
programmer 	hugo
tested by	oscat

returs the total days of the current month. e.g. 31 for january.
the function works for dates from 1970 - 2099
(*@KEY@:END_DESCRIPTION*)
FUNCTION DAYS_IN_MONTH:INT

(*Group:Default*)

VAR_INPUT
	IDATE :	UDINT;
END_VAR

(*@KEY@: WORKSHEET
NAME: DAYS_IN_MONTH
IEC_LANGUAGE: ST
*)
DAYS_IN_MONTH := DAY_OF_YEAR(IDATE);
IF LEAP_OF_DATE(IDATE) THEN
	CASE DAYS_IN_MONTH OF
		32..60	:	DAYS_IN_MONTH := 29;
		92..121 :	DAYS_IN_MONTH := 30;
		153..182:	DAYS_IN_MONTH := 30;
		245..274:	DAYS_IN_MONTH := 30;
		306..335:	DAYS_IN_MONTH := 30;
	ELSE
		DAYS_IN_MONTH := 31;
	END_CASE;
ELSE
	CASE DAYS_IN_MONTH OF
		32..59	:	DAYS_IN_MONTH := 28;
		91..120 :	DAYS_IN_MONTH := 30;
		152..181:	DAYS_IN_MONTH := 30;
		244..273:	DAYS_IN_MONTH := 30;
		305..334:	DAYS_IN_MONTH := 30;
	ELSE
		DAYS_IN_MONTH := 31;
	END_CASE;
END_IF;

(* revision history
hm	27. mar. 2009		rev 1.0
	original version

*)
(*@KEY@: END_WORKSHEET *)
END_FUNCTION

(* ---- DAYS_IN_YEAR.ST ---- *)
(*@PROPERTIES_EX@
TYPE: POU
LOCALE: 0
IEC_LANGUAGE: ST
PLC_TYPE: independent
PROC_TYPE: independent
GROUP: TIME_DATE
*)
(*@KEY@:DESCRIPTION*)
version 1.0	27. mar. 2009
programmer 	hugo
tested by	oscat

returs the total days of the year.
the function retruns 366 for leap years and 365 otherwise.
the function works for dates from 1970 - 2099
(*@KEY@:END_DESCRIPTION*)
FUNCTION DAYS_IN_YEAR:INT

(*Group:Default*)

VAR_INPUT
	IDATE :	UDINT;
END_VAR

(*@KEY@: WORKSHEET
NAME: DAYS_IN_YEAR
IEC_LANGUAGE: ST
*)
IF LEAP_OF_DATE(IDATE) THEN
	DAYS_IN_YEAR := 366;
ELSE
	DAYS_IN_YEAR := 365;
END_IF;

(* revision history
hm	27. mar. 2009		rev 1.0
	original version

*)
(*@KEY@: END_WORKSHEET *)
END_FUNCTION

(* ---- DEAD_BAND.ST ---- *)
(*@PROPERTIES_EX@
TYPE: POU
LOCALE: 0
IEC_LANGUAGE: ST
PLC_TYPE: independent
PROC_TYPE: independent
GROUP: ENGINEERING.CONTROL
*)
(*@KEY@:DESCRIPTION*)
version 1.2	18. jan. 2011
programmer 	hugo
tested by	oscat

DEAD_BAND ist eine lineare Übertragungsfunktion mit Totzone. Die Funktion verschiebt den positiven Teil der Kurve um +L und den negativen Teil der Kurve um -L.
DEAD_BAND = X - L wenn X > L)
DEAD_BAND = X + L wenn X < -L
DEAD_BAND = 0 wenn Abs(X) <= L

(*@KEY@:END_DESCRIPTION*)
FUNCTION DEAD_BAND:REAL

(*Group:Default*)

VAR_INPUT
	X :	REAL;
	L :	REAL;
END_VAR

(*@KEY@: WORKSHEET
NAME: DEAD_BAND
IEC_LANGUAGE: ST
*)
IF X > L THEN
	DEAD_BAND := X - L;
ELSIF X < -L THEN
	DEAD_BAND := X + L;
ELSE
	DEAD_BAND := 0.0;
END_IF;

(* revision history
hm	2. nov. 2007	rev 1.0
	original version

hm	14. jun. 2008	rev 1.1
	improved performance

hm	18. jan. 2011	rev 1.2
	assign 0 before return
*)
(*@KEY@: END_WORKSHEET *)
END_FUNCTION

(* ---- DEAD_ZONE.ST ---- *)
(*@PROPERTIES_EX@
TYPE: POU
LOCALE: 0
IEC_LANGUAGE: ST
PLC_TYPE: independent
PROC_TYPE: independent
GROUP: ENGINEERING.CONTROL
*)
(*@KEY@:DESCRIPTION*)
version 1.2	11. mar. 2009
programmer 	hugo
tested by	oscat

dead_zone2 is a linear transfer function which follows a linear function except for x is close to 0.
Y = X if abs(x) > L otherwise its 0.

(*@KEY@:END_DESCRIPTION*)
FUNCTION DEAD_ZONE:REAL

(*Group:Default*)

VAR_INPUT
	X :	REAL;
	L :	REAL;
END_VAR

(*@KEY@: WORKSHEET
NAME: DEAD_ZONE
IEC_LANGUAGE: ST
*)
IF ABS(x) > L THEN
	dead_zone := X;
ELSE
	DEAD_ZONE := 0.0;
END_IF;

(* revision history
hm	12. feb. 2007	rev 1.0
	original version

hm	14. jun. 2008	rev 1.1
	improved performance

hm	11. mar. 2009	rev 1.2
	real constants updated to new systax using dot

*)
(*@KEY@: END_WORKSHEET *)
END_FUNCTION

(* ---- DEC1.ST ---- *)
(*@PROPERTIES_EX@
TYPE: POU
LOCALE: 0
IEC_LANGUAGE: ST
PLC_TYPE: independent
PROC_TYPE: independent
GROUP: MATHEMATICAL.MATHE
*)
(*@KEY@:DESCRIPTION*)
version 1.1	27. oct. 2008
programmer 	hugo
tested by	oscat

This is a decrement function which decrements the variable X by 1 and if 0 is reached, it begins with M again.
_dec1(3,X) will generate 3,2,1,0,3,2,...
(*@KEY@:END_DESCRIPTION*)
FUNCTION DEC1:INT

(*Group:Default*)

VAR_INPUT
	X :	INT;
	N :	INT;
END_VAR

(*@KEY@: WORKSHEET
NAME: DEC1
IEC_LANGUAGE: ST
*)
IF X = 0 THEN
	DEC1 := N - 1;
ELSE
	DEC1 := X - 1;
END_IF;

(* this is a very elegant version but 50% slower
X := (X - 1 + N) MOD N;
*)

(* revision history
hm	13. oct. 2008	rev 1.0
	original version

hm	27. oct. 2008	rev 1.1
	added statement to return value for compatibility reasons
*)
(*@KEY@: END_WORKSHEET *)
END_FUNCTION

(* ---- DEG.ST ---- *)
(*@PROPERTIES_EX@
TYPE: POU
LOCALE: 0
IEC_LANGUAGE: ST
PLC_TYPE: independent
PROC_TYPE: independent
GROUP: MATHEMATICAL.MATHE
*)
(*@KEY@:DESCRIPTION*)
version 1.2	10. mar. 2009
programmer 	hugo
tested by	tobias

this function converts degrees into Radiant
execution time on wago 750 - 841 =  10  us
(*@KEY@:END_DESCRIPTION*)
FUNCTION DEG:REAL

(*Group:Default*)

VAR_INPUT
	RAD :	REAL;
END_VAR

(*@KEY@: WORKSHEET
NAME: DEG
IEC_LANGUAGE: ST
*)
DEG := MODR(57.29577951308232 * RAD, 360.0);

(* revision history
hm	4. aug 2006	rev 1.0
	original version

hm 16. oct 2007	rev 1.1
	added modr statement which prohibits deg to become bigger than 360

hm	10. mar. 2009	rev 1.2
	real constants updated to new systax using dot
*)
(*@KEY@: END_WORKSHEET *)
END_FUNCTION

(* ---- DIFFER.ST ---- *)
(*@PROPERTIES_EX@
TYPE: POU
LOCALE: 0
IEC_LANGUAGE: ST
PLC_TYPE: independent
PROC_TYPE: independent
GROUP: MATHEMATICAL.MATHE
*)
(*@KEY@:DESCRIPTION*)
version 1.1	16 mar 2008
programmer 	hugo
tested by	tobias

this function checks if in1 differs more then x from in2
the output is true if abs(in1-in2) > X
(*@KEY@:END_DESCRIPTION*)
FUNCTION DIFFER:BOOL

(*Group:Default*)

VAR_INPUT
	IN1 :	REAL;
	IN2 :	REAL;
	X :	REAL;
END_VAR

(*@KEY@: WORKSHEET
NAME: DIFFER
IEC_LANGUAGE: ST
*)
DIFFER := ABS(in1 - in2) > X;

(* revision history
hm		8. oct 2006		rev 1.0
	original version

hm		16. mar 2008	rev 1.1
	improverd code for performance

*)
(*@KEY@: END_WORKSHEET *)
END_FUNCTION

(* ---- DST.ST ---- *)
(*@PROPERTIES_EX@
TYPE: POU
LOCALE: 0
IEC_LANGUAGE: ST
PLC_TYPE: independent
PROC_TYPE: independent
GROUP: TIME_DATE
*)
(*@KEY@:DESCRIPTION*)
version 1.5	24. jan. 2011
programmer 	hugo
tested by	oscat

this functions returns TRUE IF dst TIME is active
the FUNCTION calculates automatically for any year betweek 1970 AND 2099
wheather daylight savings is on OR off
the summertime calculation is done according to european standards.
dst will become TRUE AT 01:00 utc in the morning FOR the respective days
AND it will become FALSE after daylight savings TIME is switched back end OF october at 01:00 utc

(*@KEY@:END_DESCRIPTION*)
FUNCTION DST:BOOL

(*Group:Default*)

VAR_INPUT
	UTC :	UDINT;
END_VAR

VAR
	yr :	INT;
	yr4 :	UDINT;
	ltc :	UDINT;
	idate :	UDINT;
END_VAR

(*@KEY@: WORKSHEET
NAME: DST
IEC_LANGUAGE: ST
*)
yr := YEAR_OF_DATE(DT_TO_DATE(UTC));
ltc := UTC;
idate := SET_DT(yr, 3, 31, 1, 0, 0);
yr4 := DWORD_TO_UDINT(SHR(INT_TO_DWORD(5 * yr), 2)) + UDINT#1;
DST := (idate - ((yr4 + UDINT#3) MOD UDINT#7) * UDINT#86400 <= ltc) AND (idate + (UDINT#214 - (yr4) MOD UDINT#7) * UDINT#86400 > ltc);

(*
Equation used TO calculate the beginning OF European Summer TIME:
Sunday (31 - (5*y/4 + 4) mod 7) March at 01.00 UTC
(valid through 2099, courtesy of Robert H. van Gent, EC).

European Summer Time ends (clocks go back) at 01.00 UTC on

    * 29 October 2006
    * 28 October 2007
    * 26 October 2008

Equation used to calculate the end of European Summer Time:
Sunday (31 - (5*y/4 + 1) mod 7) October at 01.00 UTC
(validity AND credits as above).

*)

(* revision history
hm	4. aug 2006	rev 1.0
	original version

hm	24. okt 2007	rev 1.1
	deleted time_zone_offset input because dst is generally at 01:00 utc and not mesz
	uk starts 01:00 utc and also greece

hm	1. dec 2007	rev 1.2
	changed code to improve performance

hm	16. mar. 2008	rev 1.3
	added type conversion to avoid warnings under codesys 3.0
	code improvement for better performance

hm	7. oct. 2008	rev 1.4
	changed name of function year to year_of_date

hm	24. jan. 2011	rev 1.5
	improved performance
*)

(*@KEY@: END_WORKSHEET *)
END_FUNCTION

(* ---- DWORD_OF_BYTE.ST ---- *)
(*@PROPERTIES_EX@
TYPE: POU
LOCALE: 0
IEC_LANGUAGE: ST
PLC_TYPE: independent
PROC_TYPE: independent
GROUP: LOGIC.GATE_LOGIC
*)
(*@KEY@:DESCRIPTION*)
version 1.3	18. jul. 2009
programmer 	hugo
tested by	tobias

this function creates a Dword from 4 individual bytes
(*@KEY@:END_DESCRIPTION*)
FUNCTION DWORD_OF_BYTE:DWORD

(*Group:Default*)

VAR_INPUT
	B3 :	BYTE;
	B2 :	BYTE;
	B1 :	BYTE;
	B0 :	BYTE;
END_VAR

(*@KEY@: WORKSHEET
NAME: DWORD_OF_BYTE
IEC_LANGUAGE: ST
*)
DWORD_OF_BYTE := SHL(SHL(SHL(BYTE_TO_DWORD(B3),8) OR BYTE_TO_DWORD(B2),8) OR BYTE_TO_DWORD(B1),8) OR BYTE_TO_DWORD(B0);

(* revision history
hm	24. jan 2007	rev 1.0
	original version

hm 2. jan 2008	rev 1.1
	inproved performance

hm	23. apr. 2008	rev 1.2
	reverse order of inputs to be more logical

hm	18. jul. 2009	rev 1.3
	added type conversions for compatibility reasons
*)
(*@KEY@: END_WORKSHEET *)
END_FUNCTION

(* ---- DWORD_OF_WORD.ST ---- *)
(*@PROPERTIES_EX@
TYPE: POU
LOCALE: 0
IEC_LANGUAGE: ST
PLC_TYPE: independent
PROC_TYPE: independent
GROUP: LOGIC.GATE_LOGIC
*)
(*@KEY@:DESCRIPTION*)
version 1.0	18. jul. 2009
programmer 	hugo
tested by	tobias

this function creates a Dword from 2 individual Words
(*@KEY@:END_DESCRIPTION*)
FUNCTION DWORD_OF_WORD:DWORD

(*Group:Default*)

VAR_INPUT
	W1 :	WORD;
	W0 :	WORD;
END_VAR

(*@KEY@: WORKSHEET
NAME: DWORD_OF_WORD
IEC_LANGUAGE: ST
*)
DWORD_OF_WORD := SHL_DWORD(WORD_TO_DWORD(W1),16) OR WORD_TO_DWORD(W0);

(* revision history

hm	18. jul. 2009	rev 1.0
	original version

*)
(*@KEY@: END_WORKSHEET *)
END_FUNCTION

(* ---- EASTER.ST ---- *)
(*@PROPERTIES_EX@
TYPE: POU
LOCALE: 0
IEC_LANGUAGE: ST
PLC_TYPE: independent
PROC_TYPE: independent
GROUP: TIME_DATE
*)
(*@KEY@:DESCRIPTION*)
version 1.3	7. apr. 2008
programmer 	hugo
tested by	tobias

easter calculates the day of easter sunday for a given year.
most other catholic holidays are calculated in reference to easter sunday.
(*@KEY@:END_DESCRIPTION*)
FUNCTION EASTER:UDINT

(*Group:Default*)

VAR_INPUT
	YEAR :	INT;
END_VAR

VAR
	b :	INT;
	c :	INT;
	oday :	INT;
END_VAR

(*@KEY@: WORKSHEET
NAME: EASTER
IEC_LANGUAGE: ST
*)
b := (204 - 11 * (year MOD 19)) MOD 30;
IF b > 27 THEN b := b - 1; END_IF;
c := (year + WORD_TO_INT(SHR(INT_TO_WORD(year),2)) + b - 13) MOD 7;
oday := 28 + b - c;
IF oday > 33 THEN
	easter := set_Date(year, 4, oday - 31);
ELSE
	easter := set_Date(year, 3, oday);
END_IF;

(* alternativer algorithmus ueber das pasah fest
execution time roughly 200us
Der sog. Passah-Vollmond wird berechnet, in dem das Jahr durch 19 ge-
teilt wird und der Rest mit der folgenden Tabelle verglichen wird:

    0: Apr 14       5: Apr 18      10: Mrz 25      15: Mrz 30
    1: Apr 03       6: Apr 08      11: Apr 13      16: Apr 17
    2: Mrz 23       7: Mrz 28      12: Apr 02      17: Apr 07
    3: Apr 11       8: Apr 16      13: Mrz 22      18: Mrz 27
    4: Mrz 31       9: Apr 05      14: Apr 10

Faellt dieses Datum auf einen Sonntag, ist Ostern der naechste Sonntag!

Beispiel: 1992 MOD 19 = 16, daraus folgt 17.04., der naechste Sonntag
          ist dann der 19. April (Ostersonntag)
*)

(* this algorithm is 180 us
a := year MOD 19;
b := year / 100;
c := year MOD 100;
d := b / 4;
e := b MOD 4;
f := (b + 8) / 25;
g := (b - f + 1) / 3;
h := (19 * a + b - d -g + 15) MOD 30;
i := C / 4;
k := c MOD 4;
l := (32 + 2*e + 2*i - h - k) MOD 7;
m := (a + 11 * h + 22 * l) / 451;
x := h + l - 7 * m + 114;
n := X / 31;
o := x MOD 31 + 1;

easter := set_Date(year,n,o);
*)
(*
Im Magazin "Nature" vom 20. April 1876 veröffentlichte ein anonymer Autor eine Tabelle mit Regeln zur Berechnung des (Gregorianischen) Ostersonntages des Jahres J. In Formeln ausgedrückt erhält man das Folgende:
a	=	J mod 19
b	=	int(J / 100)
c	=	J mod 100
d	=	int(b / 4)
e	=	b mod 4
f	=	int((b + 8) / 25)
g	=	int((b - f + 1) / 3
h	=	(19 · a + b - d - g + 15) mod 30
i	=	int(c / 4)
k	=	c mod 4
l	=	(32 + 2 · e + 2 · i - h - k) mod 7
m	=	int((a + 11 · h + 22 · l) / 451)
n	=	int((h + l - 7 · m + 114) / 31)
o	=	(h + l - 7 · m + 114) mod 31

n ist hierbei die Nummer des Monats, o + 1 die Nummer des Tages auf welchen der Ostersonntag im Jahr J fällt. Dieser Algorithmus kommt ohne Hilfszahlen aus.

*)

(* revision history
hm	27. dec 2006	rev 1.0
	original version

hm	15. dec 2007	rev 1.1
	modified code for better performance

hm	3. feb 2008		rev 1.2
	modified code for better performance

hm	7. apr. 2008	rev 1.3
	improved performance
*)
(*@KEY@: END_WORKSHEET *)
END_FUNCTION

(* ---- ELLIPSE_A.ST ---- *)
(*@PROPERTIES_EX@
TYPE: POU
LOCALE: 0
IEC_LANGUAGE: ST
PLC_TYPE: independent
PROC_TYPE: independent
GROUP: MATHEMATICAL.GEOMETRY
*)
(*@KEY@:DESCRIPTION*)
version 1.1	18. oct. 2008
programmer 	hugo
tested by	oscat

ellipse_A calculates the Area of an ellipe based on the two radians R1 and R2
(*@KEY@:END_DESCRIPTION*)
FUNCTION ELLIPSE_A:REAL

(*Group:Default*)

VAR_INPUT
	R1 :	REAL;
	R2 :	REAL;
END_VAR

(*@KEY@: WORKSHEET
NAME: ELLIPSE_A
IEC_LANGUAGE: ST
*)
ellipse_A := 3.14159265358979323846264338327950288 * R1 * R2;

(* revision histroy
hm	16. oct 2007	rev 1.0
	original version

hm	18. oct. 2008	rev 1.1
	using math constants
*)
(*@KEY@: END_WORKSHEET *)
END_FUNCTION

(* ---- ELLIPSE_C.ST ---- *)
(*@PROPERTIES_EX@
TYPE: POU
LOCALE: 0
IEC_LANGUAGE: ST
PLC_TYPE: independent
PROC_TYPE: independent
GROUP: MATHEMATICAL.GEOMETRY
*)
(*@KEY@:DESCRIPTION*)
version 1.2	10. mar. 2009
programmer 	hugo
tested by	oscat

ellipse_C calculates the circumference of an ellipe based on the two radians R1 and R2

(*@KEY@:END_DESCRIPTION*)
FUNCTION ELLIPSE_C:REAL

(*Group:Default*)

VAR_INPUT
	R1 :	REAL;
	R2 :	REAL;
END_VAR

(*@KEY@: WORKSHEET
NAME: ELLIPSE_C
IEC_LANGUAGE: ST
*)
ELLIPSE_C := 3.14159265358979323846264338327950288 * (3.0 * (R1+R2) - SQRT((3.0 * r1 + R2) * (3.0 * r2 + r1)));

(* revision histroy
hm	16. oct 2007	rev 1.0
	original version

hm	18. oct. 2008	rev 1.1
	using math constants

hm	10. mar. 2009	rev 1.2
	changed syntax of real constants to 0.0

*)
(*@KEY@: END_WORKSHEET *)
END_FUNCTION

(* ---- ERF.ST ---- *)
(*@PROPERTIES_EX@
TYPE: POU
LOCALE: 0
IEC_LANGUAGE: ST
PLC_TYPE: independent
PROC_TYPE: independent
GROUP: MATHEMATICAL.MATHE
*)
(*@KEY@:DESCRIPTION*)
version 1.3	10. mar. 2009
programmer 	hugo
tested by	tobias

this function calculates the erf (error) function.

(*@KEY@:END_DESCRIPTION*)
FUNCTION ERF:REAL

(*Group:Default*)

VAR_INPUT
	X :	REAL;
END_VAR

VAR
	x2 :	REAL;
	ax2 :	REAL;
END_VAR

(*@KEY@: WORKSHEET
NAME: ERF
IEC_LANGUAGE: ST
*)
x2 := X*X;
ax2 := 0.147 * x2 + 1.0;
ERF := SQRT(1.0 - EXP(-X2 * ((0.27323954473516 + aX2)/(ax2)))) * INT_TO_REAL(SGN(x));

(* revision history
hm	7. apr. 2008	rev 1.0
	original version

hm	30. jun. 2008	rev 1.1
	added type conversions to avoid warnings under codesys 3.0

hm	25. oct. 2008	rev 1.2
	new code using new algorithm

hm	10. mar. 2009	rev 1.3
	real constants updated to new systax using dot
*)
(*@KEY@: END_WORKSHEET *)
END_FUNCTION

(* ---- ERFC.ST ---- *)
(*@PROPERTIES_EX@
TYPE: POU
LOCALE: 0
IEC_LANGUAGE: ST
PLC_TYPE: independent
PROC_TYPE: independent
GROUP: MATHEMATICAL.MATHE
*)
(*@KEY@:DESCRIPTION*)
version 1.1	10. mar. 2009
programmer 	hugo
tested by	tobias

this function calculates the inverse erf (error) function.

(*@KEY@:END_DESCRIPTION*)
FUNCTION ERFC:REAL

(*Group:Default*)

VAR_INPUT
	X :	REAL;
END_VAR

(*@KEY@: WORKSHEET
NAME: ERFC
IEC_LANGUAGE: ST
*)
ERFC := 1.0 - ERF(X);

(* revision history
hm	7. apr. 2008	rev 1.0
	original version

hm	10. mar. 2009	rev 1.1
	real constants updated to new systax using dot

*)
(*@KEY@: END_WORKSHEET *)
END_FUNCTION

(* ---- EVEN.ST ---- *)
(*@PROPERTIES_EX@
TYPE: POU
LOCALE: 0
IEC_LANGUAGE: ST
PLC_TYPE: independent
PROC_TYPE: independent
GROUP: MATHEMATICAL.MATHE
*)
(*@KEY@:DESCRIPTION*)
version 1.1	1 dec 2007
programmer 	hugo
tested by	tobias

this function chacks an input for even  value
the output is true if the input is even.
(*@KEY@:END_DESCRIPTION*)
FUNCTION EVEN:BOOL

(*Group:Default*)

VAR_INPUT
	IN :	DINT;
END_VAR

(*@KEY@: WORKSHEET
NAME: EVEN
IEC_LANGUAGE: ST
*)
even := NOT BIT_OF_DWORD(DINT_TO_DWORD(in),0);

(* revision history
hm	1. oct 2006	rev 1.0
	ORIGINAL VERSION

hm	01.12.2007	rev 1.1
	changed code for improved performance

hm	21. mar. 2008	rev 1.2
	changed type of input IN from INT to DINT
*)
(*@KEY@: END_WORKSHEET *)
END_FUNCTION

(* ---- EXP10.ST ---- *)
(*@PROPERTIES_EX@
TYPE: POU
LOCALE: 0
IEC_LANGUAGE: ST
PLC_TYPE: independent
PROC_TYPE: independent
GROUP: MATHEMATICAL.MATHE
*)
(*@KEY@:DESCRIPTION*)
version 1.0	 2 dec 2007
programmer 	hugo
tested by	tobias

this function calculates the exponent to the basis 10
exp10(3) = 1000
(*@KEY@:END_DESCRIPTION*)
FUNCTION EXP10:REAL

(*Group:Default*)

VAR_INPUT
	X :	REAL;
END_VAR

(*@KEY@: WORKSHEET
NAME: EXP10
IEC_LANGUAGE: ST
*)
exp10 := EXP(X * 2.30258509299405);

(* revision history
hm	2. dec 2007		rev 1.0
	original version

*)
(*@KEY@: END_WORKSHEET *)
END_FUNCTION

(* ---- EXPN.ST ---- *)
(*@PROPERTIES_EX@
TYPE: POU
LOCALE: 0
IEC_LANGUAGE: ST
PLC_TYPE: independent
PROC_TYPE: independent
GROUP: MATHEMATICAL.MATHE
*)
(*@KEY@:DESCRIPTION*)
version 1.2	10. mar. 2009
programmer 	hugo
tested by	oscat

this function calculates X to the power of N (Y = X^N) whilke N is an integer
especially on CPU's without a floating point unit this algorythm is about 30 times faster then the IEC standard EXPT() Function

(*@KEY@:END_DESCRIPTION*)
FUNCTION EXPN:REAL

(*Group:Default*)

VAR_INPUT
	X :	REAL;
	N :	INT;
END_VAR

VAR
	N_word :	WORD;
	X_tmp :	REAL;
	sign :	BOOL;
END_VAR

(*@KEY@: WORKSHEET
NAME: EXPN
IEC_LANGUAGE: ST
*)
N_word := INT_TO_WORD(N);
X_tmp := X;
sign := BIT_OF_DWORD(WORD_TO_DWORD(N_word),15);
N_word := INT_TO_WORD(ABS(N));
IF BIT_OF_DWORD(WORD_TO_DWORD(N_word),0) THEN expn := X_tmp; ELSE expn := 1.0; END_IF;    (* N_word.X0 *)
N_word := SHR(N_word,1);
WHILE N_word > WORD#0 DO
	X_tmp := X_tmp * X_tmp;
	IF BIT_OF_DWORD(WORD_TO_DWORD(N_word),0) THEN expn := expn * X_tmp; END_IF;       (* N_word.X0 *)
	N_word := SHR(N_word,1);
END_WHILE;
IF sign THEN EXPN := 1.0 / EXPN; END_IF;

(* revision history
hm	4. dec 2007	rev 1.0
	original version

hm	22. oct. 2008	rev 1.1
	optimized code

hm	10. mar. 2009	rev 1.2
	removed nested comments
	real constants updated to new systax using dot

*)
(*@KEY@: END_WORKSHEET *)
END_FUNCTION

(* ---- F_LIN.ST ---- *)
(*@PROPERTIES_EX@
TYPE: POU
LOCALE: 0
IEC_LANGUAGE: ST
PLC_TYPE: independent
PROC_TYPE: independent
GROUP: MATHEMATICAL.FUNCTIONS
*)
(*@KEY@:DESCRIPTION*)
version 1.0	1 sep 2006
programmer 	hugo
tested by	tobias

this function calculates the linear equation f_lin = a*x + b
(*@KEY@:END_DESCRIPTION*)
FUNCTION F_LIN:REAL

(*Group:Default*)

VAR_INPUT
	X :	REAL;
	A :	REAL;
	B :	REAL;
END_VAR

(*@KEY@: WORKSHEET
NAME: F_LIN
IEC_LANGUAGE: ST
*)
F_lin := A * X + B;
(*@KEY@: END_WORKSHEET *)
END_FUNCTION

(* ---- F_LIN2.ST ---- *)
(*@PROPERTIES_EX@
TYPE: POU
LOCALE: 0
IEC_LANGUAGE: ST
PLC_TYPE: independent
PROC_TYPE: independent
GROUP: MATHEMATICAL.FUNCTIONS
*)
(*@KEY@:DESCRIPTION*)
version 1.0	1 jan 2007
programmer 	hugo
tested by	tobias

this function calculates the linear equation f_lin = a*x + b given by two points x1/y1 and x2/y2.
(*@KEY@:END_DESCRIPTION*)
FUNCTION F_LIN2:REAL

(*Group:Default*)

VAR_INPUT
	X :	REAL;
	X1 :	REAL;
	Y1 :	REAL;
	X2 :	REAL;
	Y2 :	REAL;
END_VAR

(*@KEY@: WORKSHEET
NAME: F_LIN2
IEC_LANGUAGE: ST
*)
F_LIN2 := (Y2 - Y1) / (X2 - X1) * (X - X1) + Y1;

(* revision history
hm	1. jan. 2007	rev 1.0
	original release

hm	17. dec. 2008	rev 1.1
	optimized formula

*)
(*@KEY@: END_WORKSHEET *)
END_FUNCTION

(* ---- F_POWER.ST ---- *)
(*@PROPERTIES_EX@
TYPE: POU
LOCALE: 0
IEC_LANGUAGE: ST
PLC_TYPE: independent
PROC_TYPE: independent
GROUP: MATHEMATICAL.FUNCTIONS
*)
(*@KEY@:DESCRIPTION*)
version 1.0	1 sep 2006
programmer 	hugo
tested by	tobias

this function calculates the power equation f_power = a*x^n
(*@KEY@:END_DESCRIPTION*)
FUNCTION F_POWER:REAL

(*Group:Default*)

VAR_INPUT
	A :	REAL;
	X :	REAL;
	N :	REAL;
END_VAR

(*@KEY@: WORKSHEET
NAME: F_POWER
IEC_LANGUAGE: ST
*)
f_power := a * EXPT(X,N);
(*@KEY@: END_WORKSHEET *)
END_FUNCTION

(* ---- F_QUAD.ST ---- *)
(*@PROPERTIES_EX@
TYPE: POU
LOCALE: 0
IEC_LANGUAGE: ST
PLC_TYPE: independent
PROC_TYPE: independent
GROUP: MATHEMATICAL.FUNCTIONS
*)
(*@KEY@:DESCRIPTION*)
version 1.1	18. Mar. 2011
programmer 	hugo
tested by	tobias

this function calculates the quadratic equation f_lin = a*x + b
(*@KEY@:END_DESCRIPTION*)
FUNCTION F_QUAD:REAL

(*Group:Default*)

VAR_INPUT
	X :	REAL;
	A :	REAL;
	B :	REAL;
	C :	REAL;
END_VAR

(*@KEY@: WORKSHEET
NAME: F_QUAD
IEC_LANGUAGE: ST
*)
F_QUAD :=  (A * X + B) * X + C;

(* revision history

hm	1. sep. 2006	rev 1.0
	original version

hm	18. mar. 2001	rev 1.1
	improved performance
*)

(*@KEY@: END_WORKSHEET *)
END_FUNCTION

(* ---- F_TO_C.ST ---- *)
(*@PROPERTIES_EX@
TYPE: POU
LOCALE: 0
IEC_LANGUAGE: ST
PLC_TYPE: independent
PROC_TYPE: independent
GROUP: ENGINEERING.CONVERSION
*)
(*@KEY@:DESCRIPTION*)
version 1.1	11. mar. 2009
programmer 	hugo
tested BY	tobias

this FUNCTION converts fahrenheit TO celsius

(*@KEY@:END_DESCRIPTION*)
FUNCTION F_TO_C:REAL

(*Group:Default*)

VAR_INPUT
	FAHRENHEIT :	REAL;
END_VAR

(*@KEY@: WORKSHEET
NAME: F_TO_C
IEC_LANGUAGE: ST
*)
F_TO_C := (fahrenheit - 32.0) * 0.5555555555555;

(* revision history
hm	4. aug 2006	rev 1.0
	original version

hm	11. mar. 2009	rev 1.1
	real constants updated to new systax using dot

*)
(*@KEY@: END_WORKSHEET *)
END_FUNCTION

(* ---- F_TO_OM.ST ---- *)
(*@PROPERTIES_EX@
TYPE: POU
LOCALE: 0
IEC_LANGUAGE: ST
PLC_TYPE: independent
PROC_TYPE: independent
GROUP: ENGINEERING.CONVERSION
*)
(*@KEY@:DESCRIPTION*)
version 1.1	18. oct. 2008
programmer 	hugo
tested by	oscat

this function converts frequency to Omega F
Omega = 2*PI*F
(*@KEY@:END_DESCRIPTION*)
FUNCTION F_TO_OM:REAL

(*Group:Default*)

VAR_INPUT
	F :	REAL;
END_VAR

(*@KEY@: WORKSHEET
NAME: F_TO_OM
IEC_LANGUAGE: ST
*)
F_to_OM := 6.283185307179586476 * F;

(* revision history
hm	22. jan. 2007	rev 1.0
	original version

hm	18. oct. 2008	rev 1.1
	unsing math constants

*)
(*@KEY@: END_WORKSHEET *)
END_FUNCTION

(* ---- F_TO_PT.ST ---- *)
(*@PROPERTIES_EX@
TYPE: POU
LOCALE: 0
IEC_LANGUAGE: ST
PLC_TYPE: independent
PROC_TYPE: independent
GROUP: ENGINEERING.CONVERSION
*)
(*@KEY@:DESCRIPTION*)
version 1.1	11. mar. 2009
programmer 	hugo
tested by	tobias

this function converts frequency to periode time
(*@KEY@:END_DESCRIPTION*)
FUNCTION F_TO_PT:TIME

(*Group:Default*)

VAR_INPUT
	F :	REAL;
END_VAR

(*@KEY@: WORKSHEET
NAME: F_TO_PT
IEC_LANGUAGE: ST
*)
F_TO_PT := DWORD_TO_TIME(_REAL_TO_DWORD(1.0 / F * 1000.0));

(* revision history

hm	4. aug. 2006	rev 1.0
	original version

hm	11. mar. 2009	rev 1.1
	real constants updated to new systax using dot

*)
(*@KEY@: END_WORKSHEET *)
END_FUNCTION

(* ---- FACT.ST ---- *)
(*@PROPERTIES_EX@
TYPE: POU
LOCALE: 0
IEC_LANGUAGE: ST
PLC_TYPE: independent
PROC_TYPE: independent
GROUP: MATHEMATICAL.MATHE
*)
(*@KEY@:DESCRIPTION*)
version 1.5	26. mar. 2011
programmer 	hugo
tested by	tobias

this function calculates the factorial of x

if the input is negative or higher then 12 the output will be -1.

(*@KEY@:END_DESCRIPTION*)
FUNCTION FACT:DINT

(*Group:Default*)

VAR_INPUT
	X :	INT;
END_VAR

(*@KEY@: WORKSHEET
NAME: FACT
IEC_LANGUAGE: ST
*)
CASE X OF
00: FACT := DINT#1;
01: FACT := DINT#1;
02: FACT := DINT#2;
03: FACT := DINT#6;
04: FACT := DINT#24;
05: FACT := DINT#120;
06: FACT := DINT#720;
07: FACT := DINT#5040;
08: FACT := DINT#40320;
09: FACT := DINT#362880;
10: FACT := DINT#3628800;
11: FACT := DINT#39916800;
12: FACT := DINT#479001600;
ELSE
    FACT := DINT#-1;
END_CASE;

(* revision history
hm 4.3.2007		rev 1.1
	changed a critical error where while loop was indefinite.

hm	10.12.2007	rev 1.2
	start value for i has changed to 2 for better performance

hm	10. mar 2008	rev 1.3
	changed output of fact to dint to allow bigger values

hm	27. oct. 2008	rev 1.4
	optimized code

hm	26. mar. 2011	rev 1.5
	using array math.facts
*)

(*@KEY@: END_WORKSHEET *)
END_FUNCTION

(* ---- FIB.ST ---- *)
(*@PROPERTIES_EX@
TYPE: POU
LOCALE: 0
IEC_LANGUAGE: ST
PLC_TYPE: independent
PROC_TYPE: independent
GROUP: MATHEMATICAL.MATHE
*)
(*@KEY@:DESCRIPTION*)
version 1.3	26. mar. 2008
programmer 	hugo
tested by	tobias

this function calculates the fibonacci sequence
(*@KEY@:END_DESCRIPTION*)
FUNCTION FIB:DINT

(*Group:Default*)

VAR_INPUT
	X :	INT;
END_VAR

VAR
	t1 :	DINT;
	t2 :	DINT;
	X_tmp :	INT;
END_VAR

(*@KEY@: WORKSHEET
NAME: FIB
IEC_LANGUAGE: ST
*)
t1 := DINT#0;
t2 := DINT#0;
X_tmp := X;
IF X_tmp < 0 OR X_tmp > 46 THEN
	FIB := DINT#-1;
ELSIF X_tmp < 2 THEN
	FIB := INT_TO_DINT(X_tmp);
	RETURN;
ELSE
	(* the fibonacci number is the sum of the two suceeding fibonaci numbers *)
	(* we store the numbers alternatively in t1 and t2 depending on pt *)
	t2 := DINT#1;
	WHILE X_tmp > 3 DO
		X_tmp := X_tmp - 2;
		t1 := t1 + t2;
		t2 := t1 + t2;
	END_WHILE;
	IF X_tmp > 2 THEN t1 := t1 + t2; END_IF;
	fib := t1 + t2;
END_IF;

(* alternative code for very big numbers

IF X < 31 THEN
	fib := 0.4472136 * (expn(1.618034,X) - expn(-0.618034,X));
ELSE
	fib := 0.4472133 * expn(1.618034,X);
END_IF;

*)

(* revision history
hm		27. dec 2007	rev 1.0
	original version

hm		2. jan 2008	rev 1.1
	deleted unused variable pt

hm		10. mar 2008	rev 1.2
	changed output to dint instead of real

hm		26. mar. 2008	rev 1.3
	function now returns -1 for input < 0 or > 46

*)
(*@KEY@: END_WORKSHEET *)
END_FUNCTION

(* ---- FLOOR.ST ---- *)
(*@PROPERTIES_EX@
TYPE: POU
LOCALE: 0
IEC_LANGUAGE: ST
PLC_TYPE: independent
PROC_TYPE: independent
GROUP: MATHEMATICAL.MATHE
*)
(*@KEY@:DESCRIPTION*)
version 1.1	21. mar. 2008
programmer 	hugo
tested by	tobias

This is a rounding function which returns the biggest possible integer which is less or equal to X.
floor(3.14) = 3
floor(-3.14) = -4
(*@KEY@:END_DESCRIPTION*)
FUNCTION FLOOR:INT

(*Group:Default*)

VAR_INPUT
	X :	REAL;
END_VAR

(*@KEY@: WORKSHEET
NAME: FLOOR
IEC_LANGUAGE: ST
*)
FLOOR := REAL_TO_INT(X);
IF INT_TO_REAL(FLOOR) > X THEN
	floor := floor - 1;
END_IF;

(* revision history
hm		7. feb 2007		rev 1.0
	originlal version

hm		21. mar. 2008	rev 1.1
	replaced trunc with real_to_int for compatibility reasons

*)
(*@KEY@: END_WORKSHEET *)
END_FUNCTION

(* ---- FLOOR2.ST ---- *)
(*@PROPERTIES_EX@
TYPE: POU
LOCALE: 0
IEC_LANGUAGE: ST
PLC_TYPE: independent
PROC_TYPE: independent
GROUP: MATHEMATICAL.MATHE
*)
(*@KEY@:DESCRIPTION*)
version 1.1	4. apr. 2008
programmer 	hugo
tested by	tobias

This is a rounding function which returns the biggest possible integer which is less or equal to X.
floor2(3.14) = 3
floor2(-3.14) = -4
(*@KEY@:END_DESCRIPTION*)
FUNCTION FLOOR2:DINT

(*Group:Default*)

VAR_INPUT
	X :	REAL;
END_VAR

(*@KEY@: WORKSHEET
NAME: FLOOR2
IEC_LANGUAGE: ST
*)
FLOOR2 := _REAL_TO_DINT(X);
IF DINT_TO_REAL(FLOOR2) > X THEN
	FLOOR2 := FLOOR2 - DINT#1;
END_IF;

(* revision history
hm	21. mar. 2008	rev 1.0
	originlal version

hm	4. apr. 2008	rev 1.1
	added type conversion to avoid warnings under codesys 3.0
*)
(*@KEY@: END_WORKSHEET *)
END_FUNCTION

(* ---- FRACT.ST ---- *)
(*@PROPERTIES_EX@
TYPE: POU
LOCALE: 0
IEC_LANGUAGE: ST
PLC_TYPE: independent
PROC_TYPE: independent
GROUP: MATHEMATICAL.MATHE
*)
(*@KEY@:DESCRIPTION*)
version 1.3	10. mar. 2009
programmer 	hugo
tested by	tobias

this function returns the fraction of a real number
fract(3.14) = 0.14

(*@KEY@:END_DESCRIPTION*)
FUNCTION FRACT:REAL

(*Group:Default*)

VAR_INPUT
	X :	REAL;
END_VAR

(*@KEY@: WORKSHEET
NAME: FRACT
IEC_LANGUAGE: ST
*)
IF ABS(x) < 2.0E9 THEN
	FRACT := x - DINT_TO_REAL(D_TRUNC(x));
ELSE
	FRACT := 0.0;
END_IF;

(* revision history
hm	4. aug 2006	rev 1.0
	original version

hm	11. mar 2008	rev 1.1
	added dint_to_real for compatibility reasons
	now returns 0 for number > 2e9
	changed input to x

hm	21. mar. 2008	rev 1.2
	use D_trunc instead of TRUNC for compatibility reasons

hm	10. mar. 2009	rev 1.3
	real constants updated to new systax using dot

*)
(*@KEY@: END_WORKSHEET *)
END_FUNCTION

(* ---- FRMP_B.ST ---- *)
(*@PROPERTIES_EX@
TYPE: POU
LOCALE: 0
IEC_LANGUAGE: ST
PLC_TYPE: independent
PROC_TYPE: independent
GROUP: MATHEMATICAL.FUNCTIONS
*)
(*@KEY@:DESCRIPTION*)
version 1.0		17. feb. 2011
programmer 	    hugo
tested by		oscat

this function calculates a ramp and limits the output to 0 .. 255 without overflow problems

(*@KEY@:END_DESCRIPTION*)
FUNCTION FRMP_B:BYTE

(*Group:Default*)

VAR_INPUT
	START :	BYTE;
	DIR :	BOOL;
	TD :	TIME;
	TR :	TIME;
END_VAR

(*@KEY@: WORKSHEET
NAME: FRMP_B
IEC_LANGUAGE: ST
*)
IF TD < TR THEN
	FRMP_B := MIN(UDINT_TO_BYTE(DWORD_TO_UDINT(SHL(TIME_TO_DWORD(TD), 8)) / TIME_TO_UDINT(TR)), SEL(DIR, START, USINT_TO_BYTE(USINT#255 - BYTE_TO_USINT(START))));
	IF DIR THEN
		FRMP_B := USINT_TO_BYTE(BYTE_TO_USINT(START) + BYTE_TO_USINT(FRMP_B));
	ELSE
		FRMP_B := USINT_TO_BYTE(BYTE_TO_USINT(START) - BYTE_TO_USINT(FRMP_B));
	END_IF;
ELSE
	FRMP_B := SEL(DIR, BYTE#0, BYTE#255);
END_IF;

(* revision history

17. feb. 2011	rev 1.0
	new module

*)
(*@KEY@: END_WORKSHEET *)
END_FUNCTION

(* ---- GAMMA.ST ---- *)
(*@PROPERTIES_EX@
TYPE: POU
LOCALE: 0
IEC_LANGUAGE: ST
PLC_TYPE: independent
PROC_TYPE: independent
GROUP: MATHEMATICAL.MATHE
*)
(*@KEY@:DESCRIPTION*)
version 1.3	10. mar. 2009
programmer 	hugo
tested by	oscat

this function calculates the stirling function which is an approximation for the gamma function

(*@KEY@:END_DESCRIPTION*)
FUNCTION GAMMA:REAL

(*Group:Default*)

VAR_INPUT
	X :	REAL;
END_VAR

(*@KEY@: WORKSHEET
NAME: GAMMA
IEC_LANGUAGE: ST
*)
IF x > 0.0 THEN
	GAMMA := SQRT(6.28318530717958647692528676655900576 / X) * EXPT(0.367879441171442 * (x + 1.0 / (12.0 * x - 0.1 / X)), X);
END_IF;

(* the stirling formula is not very accurate for small values of X
IF X >=0 THEN GAMMA := SQRT(math.PI2 * X) * EXPT(X / math.E, X); END_IF;
*)

(* revision history
hm	10.12.2007	rev 1.0
	original version

hm	18. oct. 2008	rev 1.1
	using math constants

hm	26. oct. 2008	rev 1.2
	using new formula with better accuracy

hm	10. mar. 2009	rev 1.3
	real constants updated to new systax using dot

*)
(*@KEY@: END_WORKSHEET *)
END_FUNCTION

(* ---- GAUSS.ST ---- *)
(*@PROPERTIES_EX@
TYPE: POU
LOCALE: 0
IEC_LANGUAGE: ST
PLC_TYPE: independent
PROC_TYPE: independent
GROUP: MATHEMATICAL.MATHE
*)
(*@KEY@:DESCRIPTION*)
version 1.2	10. mar. 2009
programmer 	hugo
tested by	tobias

this function calculates the gaussian density function

(*@KEY@:END_DESCRIPTION*)
FUNCTION GAUSS:REAL

(*Group:Default*)

VAR_INPUT
	X :	REAL;
	U :	REAL;
	SI :	REAL;
END_VAR

VAR
	temp :	REAL;
	si_inv :	REAL;
END_VAR

(*@KEY@: WORKSHEET
NAME: GAUSS
IEC_LANGUAGE: ST
*)
temp := X - U;
si_inv := 1.0  / si;
GAUSS := EXP(Temp * Temp * si_inv * SI_inv * - 0.5) * 0.39894228 * si_inv;

(* revision hisdtory
hm	6. apr. 2008	rev 1.0
	original version

hm	27. oct. 2008	rev 1.1
	optimized performance

hm	10. mar. 2009	rev 1.2
	real constants updated to new systax using dot

*)
(*@KEY@: END_WORKSHEET *)
END_FUNCTION

(* ---- GAUSSCD.ST ---- *)
(*@PROPERTIES_EX@
TYPE: POU
LOCALE: 0
IEC_LANGUAGE: ST
PLC_TYPE: independent
PROC_TYPE: independent
GROUP: MATHEMATICAL.MATHE
*)
(*@KEY@:DESCRIPTION*)
version 1.1	10. mar. 2009
programmer 	hugo
tested by	tobias

this function calculates the gaussian cumulative distribution function

(*@KEY@:END_DESCRIPTION*)
FUNCTION GAUSSCD:REAL

(*Group:Default*)

VAR_INPUT
	X :	REAL;
	U :	REAL;
	SI :	REAL;
END_VAR

(*@KEY@: WORKSHEET
NAME: GAUSSCD
IEC_LANGUAGE: ST
*)
GAUSSCD := (ERF((X - U) / (SI * 1.414213562)) + 1.0) * 0.5;

(* revision hisdtory
hm	6. apr. 2008	rev 1.0
	original version

hm	10. mar. 2009	rev 1.1
	real constants updated to new systax using dot

*)

(*@KEY@: END_WORKSHEET *)
END_FUNCTION

(* ---- GCD.ST ---- *)
(*@PROPERTIES_EX@
TYPE: POU
LOCALE: 0
IEC_LANGUAGE: ST
PLC_TYPE: independent
PROC_TYPE: independent
GROUP: MATHEMATICAL.MATHE
*)
(*@KEY@:DESCRIPTION*)
version 1.0	19. jan. 2011
programmer 	hugo
tested by	tobias

this function calculates the gretaest common divisor of two numbers A and B

(*@KEY@:END_DESCRIPTION*)
FUNCTION GCD:INT

(*Group:Default*)

VAR_INPUT
	A :	DINT;
	B :	DINT;
END_VAR

VAR
	t :	DINT;
	_A :	DINT;
	_B :	DINT;
END_VAR

(*@KEY@: WORKSHEET
NAME: GCD
IEC_LANGUAGE: ST
*)
_A := A;
_B := B;

IF _A = DINT#0 THEN
	GCD := DINT_TO_INT(ABS(_B));
ELSIF _B = DINT#0 THEN
	GCD := DINT_TO_INT(ABS(_A));
ELSE
	_A := ABS(_A);
	_B := ABS(_B);
	GCD := 1;

	WHILE NOT((DINT_TO_DWORD(_A) AND DWORD#1) > DWORD#0 OR (DINT_TO_DWORD(_B) AND DWORD#1) > DWORD#0) DO
		_A := DWORD_TO_DINT(SHR(DINT_TO_DWORD(_A),1));
		_B := DWORD_TO_DINT(SHR(DINT_TO_DWORD(_B),1));
		GCD := DWORD_TO_INT(SHR(INT_TO_DWORD(GCD),1));
	END_WHILE;
	WHILE _A > DINT#0 DO
		IF NOT((DINT_TO_DWORD(_A) AND DWORD#1) > DWORD#0) THEN
			_A := DWORD_TO_DINT(SHR(DINT_TO_DWORD(_A),1));
		ELSIF NOT((DINT_TO_DWORD(_B) AND DWORD#1) > DWORD#0) THEN
			_B := DWORD_TO_DINT(SHR(DINT_TO_DWORD(_B),1));
		ELSE
			t := DWORD_TO_DINT(SHR(DINT_TO_DWORD(ABS(_A-_B)),1));
			IF _A < _B THEN
				_B := t;
			ELSE
				_A := t;
			END_IF;
		END_IF;
	END_WHILE;
	GCD := GCD * DINT_TO_INT(_B);
END_IF;

(* revision history
hm	19. jan. 2011	rev 1.0
	original version

*)

(*@KEY@: END_WORKSHEET *)
END_FUNCTION

(* ---- GDF.ST ---- *)
(*@PROPERTIES_EX@
TYPE: POU
LOCALE: 0
IEC_LANGUAGE: ST
PLC_TYPE: independent
PROC_TYPE: independent
GROUP: MATHEMATICAL.MATHE
*)
(*@KEY@:DESCRIPTION*)
version 1.2	10. mar. 2009
programmer 	hugo
tested by	tobias

this function calculates the Gudermannian function.
(*@KEY@:END_DESCRIPTION*)
FUNCTION GDF:REAL

(*Group:Default*)

VAR_INPUT
	X :	REAL;
END_VAR

(*@KEY@: WORKSHEET
NAME: GDF
IEC_LANGUAGE: ST
*)
IF X = 0.0 THEN
	GDF := 0.0;
ELSIF X > 15.0 THEN
	GDF := 1.5707963267949;
ELSIF X < -15.0 THEN
	GDF := -1.5707963267949;
ELSE
	GDF := ATAN(EXP(X)) * 2.0 - 1.5707963267949;
END_IF;

(* revision history
hm	27. apr. 2008	rev 1.0
	original version

hm	18. oct. 2008	rev 1.1
	using math constants

hm	10. mar. 2009	rev 1.2
	real constants updated to new systax using dot

*)

(*@KEY@: END_WORKSHEET *)
END_FUNCTION

(* ---- GEO_TO_DEG.ST ---- *)
(*@PROPERTIES_EX@
TYPE: POU
LOCALE: 0
IEC_LANGUAGE: ST
PLC_TYPE: independent
PROC_TYPE: independent
GROUP: ENGINEERING.CONVERSION
*)
(*@KEY@:DESCRIPTION*)
version 1.0	22. jan. 2009
programmer 	hugo
tested by	oscat

this function converts degrees, minutes seconds to decimal degrees.
(*@KEY@:END_DESCRIPTION*)
FUNCTION GEO_TO_DEG:REAL

(*Group:Default*)

VAR_INPUT
	D :	INT;
	M :	INT;
	SEC :	REAL;
END_VAR

(*@KEY@: WORKSHEET
NAME: GEO_TO_DEG
IEC_LANGUAGE: ST
*)
GEO_TO_DEG := INT_TO_REAL(D) + INT_TO_REAL(M) * 0.016666666666667 + sec * 0.00027777777777778;

(* revision histroy
hm	22. jan. 2009	rev 1.0
	original release

*)
(*@KEY@: END_WORKSHEET *)
END_FUNCTION

(* ---- GOLD.ST ---- *)
(*@PROPERTIES_EX@
TYPE: POU
LOCALE: 0
IEC_LANGUAGE: ST
PLC_TYPE: independent
PROC_TYPE: independent
GROUP: MATHEMATICAL.MATHE
*)
(*@KEY@:DESCRIPTION*)
version 1.1	10. mar. 2009
programmer 	hugo
tested by	tobias

this function calculates the golden function.

(*@KEY@:END_DESCRIPTION*)
FUNCTION GOLD:REAL

(*Group:Default*)

VAR_INPUT
	X :	REAL;
END_VAR

(*@KEY@: WORKSHEET
NAME: GOLD
IEC_LANGUAGE: ST
*)
GOLD := (X + SQRT(X*X + 4.0)) * 0.5;

(* revision history
hm	27. apr. 2008	rev 1.0
	original version

hm	10. mar. 2009	rev 1.1
	real constants updated to new systax using dot

*)
(*@KEY@: END_WORKSHEET *)
END_FUNCTION

(* ---- GRAY_TO_BYTE.ST ---- *)
(*@PROPERTIES_EX@
TYPE: POU
LOCALE: 0
IEC_LANGUAGE: ST
PLC_TYPE: independent
PROC_TYPE: independent
GROUP: LOGIC.GATE_LOGIC
*)
(*@KEY@:DESCRIPTION*)
version 1.0	9. nov. 2009
programmer 	hugo
tested by	oscat

this function converts a gray code into binary

(*@KEY@:END_DESCRIPTION*)
FUNCTION GRAY_TO_BYTE:BYTE

(*Group:Default*)

VAR_INPUT
	IN :	BYTE;
END_VAR

(*@KEY@: WORKSHEET
NAME: GRAY_TO_BYTE
IEC_LANGUAGE: ST
*)
GRAY_TO_BYTE := SHR_BYTE(IN,4) XOR IN;
GRAY_TO_BYTE := SHR_BYTE(GRAY_TO_BYTE,2) XOR GRAY_TO_BYTE;
GRAY_TO_BYTE := SHR_BYTE(GRAY_TO_BYTE,1) XOR GRAY_TO_BYTE;

(* revision history
hm	9. nov. 2009	rev 1.0
	original version

*)

(*@KEY@: END_WORKSHEET *)
END_FUNCTION

(* ---- HOUR.ST ---- *)
(*@PROPERTIES_EX@
TYPE: POU
LOCALE: 0
IEC_LANGUAGE: ST
PLC_TYPE: independent
PROC_TYPE: independent
GROUP: TIME_DATE
*)
(*@KEY@:DESCRIPTION*)
version 1.1	2 okt 2006
programmer 	hugo
tested by	tobias

extracts the hour of a Time_of_day
(*@KEY@:END_DESCRIPTION*)
FUNCTION HOUR:INT

(*Group:Default*)

VAR_INPUT
	ITOD :	UDINT;
END_VAR

(*@KEY@: WORKSHEET
NAME: HOUR
IEC_LANGUAGE: ST
*)
hour := UDINT_TO_INT(itod / UDINT#3600000);

(* change history
hm 4. aug 2006	rev 1.0
	original version

hm 2.10.2006 	rev 1.1
	changed name of input to itod

*)
(*@KEY@: END_WORKSHEET *)
END_FUNCTION

(* ---- HOUR_OF_DT.ST ---- *)
(*@PROPERTIES_EX@
TYPE: POU
LOCALE: 0
IEC_LANGUAGE: ST
PLC_TYPE: independent
PROC_TYPE: independent
GROUP: TIME_DATE
*)
(*@KEY@:DESCRIPTION*)
version 1.0	6. jun. 2008
programmer 	oscat
tested BY	oscat

HOUR_OF_DT returns the current hour (hour of the day) of a DT variable
(*@KEY@:END_DESCRIPTION*)
FUNCTION HOUR_OF_DT:INT

(*Group:Default*)

VAR_INPUT
	XDT :	UDINT;
END_VAR

(*@KEY@: WORKSHEET
NAME: HOUR_OF_DT
IEC_LANGUAGE: ST
*)
HOUR_OF_DT := UDINT_TO_INT((XDT MOD UDINT#86400) / UDINT#3600);

(* revision history
hm		6.9.2008	rev 1.0
	original version

*)
(*@KEY@: END_WORKSHEET *)
END_FUNCTION

(* ---- HOUR_TO_TIME.ST ---- *)
(*@PROPERTIES_EX@
TYPE: POU
LOCALE: 0
IEC_LANGUAGE: ST
PLC_TYPE: independent
PROC_TYPE: independent
GROUP: TIME_DATE
*)
(*@KEY@:DESCRIPTION*)
version 1.2	24. feb. 2009
programmer 	hugo
tested by	tobias

converts an amount of hours in real to time
(*@KEY@:END_DESCRIPTION*)
FUNCTION HOUR_TO_TIME:TIME

(*Group:Default*)

VAR_INPUT
	IN :	REAL;
END_VAR

(*@KEY@: WORKSHEET
NAME: HOUR_TO_TIME
IEC_LANGUAGE: ST
*)
hour_to_time := UDINT_TO_TIME(_REAL_TO_UDINT(IN * 3600000.0));

(* revision history
hm		4. aug 2006	rev 1.0
	original version

hm		14. mar 2008	rev 1.1
	rounded the input after the last digit

*)
(*@KEY@: END_WORKSHEET *)
END_FUNCTION

(* ---- HOUR_TO_TOD.ST ---- *)
(*@PROPERTIES_EX@
TYPE: POU
LOCALE: 0
IEC_LANGUAGE: ST
PLC_TYPE: independent
PROC_TYPE: independent
GROUP: TIME_DATE
*)
(*@KEY@:DESCRIPTION*)
version 1.1	14 aug 2008
programmer 	hugo
tested by	tobias

converts an amount of hours in real to time of day TOD.
(*@KEY@:END_DESCRIPTION*)
FUNCTION HOUR_TO_TOD:UDINT

(*Group:Default*)

VAR_INPUT
	IN :	REAL;
END_VAR

(*@KEY@: WORKSHEET
NAME: HOUR_TO_TOD
IEC_LANGUAGE: ST
*)
hour_to_tod := _REAL_TO_UDINT(IN * 3600000.00);

(* revision history
hm		4. aug 2006	rev 1.0
	original version

hm		14. mar 2008	rev 1.1
	rounded the input after the last digit

*)
(*@KEY@: END_WORKSHEET *)
END_FUNCTION

(* ---- HYPOT.ST ---- *)
(*@PROPERTIES_EX@
TYPE: POU
LOCALE: 0
IEC_LANGUAGE: ST
PLC_TYPE: independent
PROC_TYPE: independent
GROUP: MATHEMATICAL.MATHE
*)
(*@KEY@:DESCRIPTION*)
version 1.0	21 feb 2008
programmer 	hugo
tested by	oscat

this function calculates the pythagorean function
es the arcus cos hyperbolicus
(*@KEY@:END_DESCRIPTION*)
FUNCTION HYPOT:REAL

(*Group:Default*)

VAR_INPUT
	X :	REAL;
	Y :	REAL;
END_VAR

(*@KEY@: WORKSHEET
NAME: HYPOT
IEC_LANGUAGE: ST
*)
HYPOT := SQRT(x*x + y*y);

(* revision history
hm	21. feb 2008	rev 1.0
	original version

*)
(*@KEY@: END_WORKSHEET *)
END_FUNCTION

(* ---- INC.ST ---- *)
(*@PROPERTIES_EX@
TYPE: POU
LOCALE: 0
IEC_LANGUAGE: ST
PLC_TYPE: independent
PROC_TYPE: independent
GROUP: MATHEMATICAL.MATHE
*)
(*@KEY@:DESCRIPTION*)
version 1.1	15. jan 2008
programmer 	hugo
tested by	tobias

This is a increment function which increments the input X by the value D and compares the result with M.
if the output exceeds M it will continue to count from 0 again.
(*@KEY@:END_DESCRIPTION*)
FUNCTION INC:INT

(*Group:Default*)

VAR_INPUT
	X :	INT;
	D :	INT;
	M :	INT;
END_VAR

(*@KEY@: WORKSHEET
NAME: INC
IEC_LANGUAGE: ST
*)
inc := (X + D + M + 1) MOD (M + 1);

(* revision history
hm	7. feb 2007		REV 1.0
	original version

hm	15. jan 2008	rev 1.1
	allow for neagtive increment

*)
(*@KEY@: END_WORKSHEET *)
END_FUNCTION

(* ---- INC1.ST ---- *)
(*@PROPERTIES_EX@
TYPE: POU
LOCALE: 0
IEC_LANGUAGE: ST
PLC_TYPE: independent
PROC_TYPE: independent
GROUP: MATHEMATICAL.MATHE
*)
(*@KEY@:DESCRIPTION*)
version 1.2	23. feb. 2009
programmer 	hugo
tested by	oscat

This is a increment function which increments the variable X by 1 and if N is reached, it begins with 0 instead of N again.
inc1(X,3) will generate 0,1,2,0,1,.....
(*@KEY@:END_DESCRIPTION*)
FUNCTION INC1:INT

(*Group:Default*)

VAR_INPUT
	X :	INT;
	N :	INT;
END_VAR

(*@KEY@: WORKSHEET
NAME: INC1
IEC_LANGUAGE: ST
*)
IF X >= N - 1 THEN
	INC1 := 0;
ELSE
	INC1 := X + 1;
END_IF;

(* this elegant version is 50% slower
INC1 := X := (x + 1) MOD N;
*)

(* revision history
hm	13. oct. 2008	rev 1.0
	original version

hm	22. oct. 2008	rev 1.1
	added statement to return value for compatibility reasons

hm	23. feb. 2009	rev 1.2
 	when inc1 is called with X >= N inc will continue with 0
*)
(*@KEY@: END_WORKSHEET *)
END_FUNCTION

(* ---- INC2.ST ---- *)
(*@PROPERTIES_EX@
TYPE: POU
LOCALE: 0
IEC_LANGUAGE: ST
PLC_TYPE: independent
PROC_TYPE: independent
GROUP: MATHEMATICAL.MATHE
*)
(*@KEY@:DESCRIPTION*)
version 1.0	29. jun. 2008
programmer 	hugo
tested by	oscat

This function increments the input X by the value D and compares the result with U.
if the output exceeds U it will continue to count from L again.
(*@KEY@:END_DESCRIPTION*)
FUNCTION INC2:INT

(*Group:Default*)

VAR_INPUT
	X :	INT;
	D :	INT;
	L :	INT;
	U :	INT;
END_VAR

VAR
	tmp :	INT;
END_VAR

(*@KEY@: WORKSHEET
NAME: INC2
IEC_LANGUAGE: ST
*)
tmp := U - L + 1;
INC2 := (X + D - L + tmp) MOD tmp + L;

(* revision history
hm	29. jun. 2008		REV 1.0
	original version

*)
(*@KEY@: END_WORKSHEET *)
END_FUNCTION

(* ---- INT_TO_BCDC.ST ---- *)
(*@PROPERTIES_EX@
TYPE: POU
LOCALE: 0
IEC_LANGUAGE: ST
PLC_TYPE: independent
PROC_TYPE: independent
GROUP: LOGIC.GATE_LOGIC
*)
(*@KEY@:DESCRIPTION*)
version 1.1	30. jun. 2008
programmer 	hugo
tested by	tobias

this function converts an integer into a two digit bcd number.
(*@KEY@:END_DESCRIPTION*)
FUNCTION INT_TO_BCDC:BYTE

(*Group:Default*)

VAR_INPUT
	IN :	INT;
END_VAR

(*@KEY@: WORKSHEET
NAME: INT_TO_BCDC
IEC_LANGUAGE: ST
*)
INT_TO_BCDC := SHL_BYTE(INT_TO_BYTE(IN / INT#10),4) OR INT_TO_BYTE(in MOD INT#10);

(* revision history
hm	13.12.2007
	original version

hm	30.6.2008	rev 1.1
	changed name INT_TO_BCD to INT_TO_BCDC to avoid collision with util.lib
	corrected error in code

*)
(*@KEY@: END_WORKSHEET *)
END_FUNCTION

(* ---- INV.ST ---- *)
(*@PROPERTIES_EX@
TYPE: POU
LOCALE: 0
IEC_LANGUAGE: ST
PLC_TYPE: independent
PROC_TYPE: independent
GROUP: MATHEMATICAL.MATHE
*)
(*@KEY@:DESCRIPTION*)
version 1.1	10. mar. 2009
programmer 	hugo
tested by	tobias

This function calculates the result of 1 / X
(*@KEY@:END_DESCRIPTION*)
FUNCTION INV:REAL

(*Group:Default*)

VAR_INPUT
	X :	REAL;
END_VAR

(*@KEY@: WORKSHEET
NAME: INV
IEC_LANGUAGE: ST
*)
IF X <> 0.0 THEN INV := 1.0 / X; END_IF;

(* revision history
hm	26. oct. 2008	rev 1.0
	original version

hm	10. mar. 2009	rev 1.1
	real constants updated to new systax using dot

*)

(*@KEY@: END_WORKSHEET *)
END_FUNCTION

(* ---- ISC_ALPHA.ST ---- *)
(*@PROPERTIES_EX@
TYPE: POU
LOCALE: 0
IEC_LANGUAGE: ST
PLC_TYPE: independent
PROC_TYPE: independent
GROUP: STRINGS
*)
(*@KEY@:DESCRIPTION*)
version 1.1	19. oct. 2008
programmer 	oscat
tested by	oscat

ISC_ALPHA checks if a character is a..z or A..Z.
(*@KEY@:END_DESCRIPTION*)
FUNCTION ISC_ALPHA:BOOL

(*Group:Default*)

VAR_INPUT
	IN :	BYTE;
END_VAR

(*@KEY@: WORKSHEET
NAME: ISC_ALPHA
IEC_LANGUAGE: ST
*)
IF SETUP_EXTENDED_ASCII(FALSE) THEN
	ISC_ALPHA := (in > BYTE#64 AND in < BYTE#91) OR (in > BYTE#191  AND in <> BYTE#215 AND in <> BYTE#247) OR (in > BYTE#96 AND in < BYTE#123);
ELSE
	ISC_ALPHA := (IN > BYTE#64 AND IN < BYTE#91) OR (in > BYTE#96 AND in < BYTE#123);
END_IF;

(* revision history
hm	6. mar. 2008	rev 1.0
	original version

hm	19. oct. 2008	rev 1.1
	changes setup constants
*)
(*@KEY@: END_WORKSHEET *)
END_FUNCTION

(* ---- ISC_CTRL.ST ---- *)
(*@PROPERTIES_EX@
TYPE: POU
LOCALE: 0
IEC_LANGUAGE: ST
PLC_TYPE: independent
PROC_TYPE: independent
GROUP: STRINGS
*)
(*@KEY@:DESCRIPTION*)
version 1.0	6. mar 2008
programmer 	oscat
tested by	hugo

ISC_ALPHA checks if a character is a control character.
(*@KEY@:END_DESCRIPTION*)
FUNCTION ISC_CTRL:BOOL

(*Group:Default*)

VAR_INPUT
	IN :	BYTE;
END_VAR

(*@KEY@: WORKSHEET
NAME: ISC_CTRL
IEC_LANGUAGE: ST
*)
ISC_CTRL := IN < BYTE#32 OR IN = BYTE#127;

(* revision history
hm		6. mar. 2008	rev 1.0
	original version

*)
(*@KEY@: END_WORKSHEET *)
END_FUNCTION

(* ---- ISC_HEX.ST ---- *)
(*@PROPERTIES_EX@
TYPE: POU
LOCALE: 0
IEC_LANGUAGE: ST
PLC_TYPE: independent
PROC_TYPE: independent
GROUP: STRINGS
*)
(*@KEY@:DESCRIPTION*)
version 1.0	6. mar 2008
programmer 	oscat
tested by		hugo

ISC_HEX checks if a character is 0..9, A..F, a..f.
(*@KEY@:END_DESCRIPTION*)
FUNCTION ISC_HEX:BOOL

(*Group:Default*)

VAR_INPUT
	IN :	BYTE;
END_VAR

(*@KEY@: WORKSHEET
NAME: ISC_HEX
IEC_LANGUAGE: ST
*)
ISC_HEX := (IN > BYTE#47 AND IN < BYTE#58) OR (IN > BYTE#64 AND IN < BYTE#71) OR (IN > BYTE#96 AND IN < BYTE#103);

(* revision history
hm		6. mar. 2008	rev 1.0
	original version

*)
(*@KEY@: END_WORKSHEET *)
END_FUNCTION

(* ---- ISC_LOWER.ST ---- *)
(*@PROPERTIES_EX@
TYPE: POU
LOCALE: 0
IEC_LANGUAGE: ST
PLC_TYPE: independent
PROC_TYPE: independent
GROUP: STRINGS
*)
(*@KEY@:DESCRIPTION*)
version 1.1	19. oct. 2008
programmer 	hugo
tested by	oscat

isc_lower checks if a character is lowercase.
(*@KEY@:END_DESCRIPTION*)
FUNCTION ISC_LOWER:BOOL

(*Group:Default*)

VAR_INPUT
	IN :	BYTE;
END_VAR

(*@KEY@: WORKSHEET
NAME: ISC_LOWER
IEC_LANGUAGE: ST
*)
IF SETUP_EXTENDED_ASCII(FALSE) THEN
	ISC_LOWER := ((in > BYTE#96) AND (in < BYTE#123)) OR ((in > BYTE#222) AND (in <> BYTE#247));
ELSE
	ISC_LOWER := ((in > BYTE#96) AND (in < BYTE#123));
END_IF;

(* revision history
hm	6. mar. 2008	rev 1.0
	original version

hm	19. oct. 2008	rev 1.1
	changes setup constants
*)
(*@KEY@: END_WORKSHEET *)
END_FUNCTION

(* ---- ISC_NUM.ST ---- *)
(*@PROPERTIES_EX@
TYPE: POU
LOCALE: 0
IEC_LANGUAGE: ST
PLC_TYPE: independent
PROC_TYPE: independent
GROUP: STRINGS
*)
(*@KEY@:DESCRIPTION*)
version 1.0	6. mar 2008
programmer 	oscat
tested by	hugo

ISC_NUM checks if a character is 0..9.
(*@KEY@:END_DESCRIPTION*)
FUNCTION ISC_NUM:BOOL

(*Group:Default*)

VAR_INPUT
	IN :	BYTE;
END_VAR

(*@KEY@: WORKSHEET
NAME: ISC_NUM
IEC_LANGUAGE: ST
*)
ISC_NUM := IN > BYTE#47 AND IN < BYTE#58;

(* revision history
hm		6. mar. 2008	rev 1.0
	original version

*)
(*@KEY@: END_WORKSHEET *)
END_FUNCTION

(* ---- ISC_UPPER.ST ---- *)
(*@PROPERTIES_EX@
TYPE: POU
LOCALE: 0
IEC_LANGUAGE: ST
PLC_TYPE: independent
PROC_TYPE: independent
GROUP: STRINGS
*)
(*@KEY@:DESCRIPTION*)
version 1.1	19. oct. 2008
programmer 	hugo
tested by	oscat

ISC_upper checks if a character is uppercase
(*@KEY@:END_DESCRIPTION*)
FUNCTION ISC_UPPER:BOOL

(*Group:Default*)

VAR_INPUT
	IN :	BYTE;
END_VAR

(*@KEY@: WORKSHEET
NAME: ISC_UPPER
IEC_LANGUAGE: ST
*)
IF SETUP_EXTENDED_ASCII(FALSE) THEN
	ISC_UPPER :=  ((in > BYTE#64) AND (in < BYTE#91)) OR (((in > BYTE#191) AND (in < BYTE#223)) AND (in <> BYTE#215));
ELSE
	ISC_UPPER := ((in > BYTE#64) AND (in < BYTE#91));
END_IF;

(* revision history
hm	6. mar. 2008	rev 1.0
	original version

hm	19. oct. 2008	rev 1.1
	changes setup constants

*)
(*@KEY@: END_WORKSHEET *)
END_FUNCTION

(* ---- JD2000.ST ---- *)
(*@PROPERTIES_EX@
TYPE: POU
LOCALE: 0
IEC_LANGUAGE: ST
PLC_TYPE: independent
PROC_TYPE: independent
GROUP: TIME_DATE
*)
(*@KEY@:DESCRIPTION*)
version 1.0	15. jul. 2008
programmer 	hugo
tested by	oscat

JULIAN calculates the astronomic julian date from 1.1.2000-12:00.

(*@KEY@:END_DESCRIPTION*)
FUNCTION JD2000:REAL

(*Group:Default*)

VAR_INPUT
	DTI :	UDINT;
END_VAR

(*@KEY@: WORKSHEET
NAME: JD2000
IEC_LANGUAGE: ST
*)
JD2000 := UDINT_TO_REAL(DTI - UDINT#946728000) / 86400.0;

(* revision histroy
hm	15. jul. 2008	rev 1.0
	original release
*)
(*@KEY@: END_WORKSHEET *)
END_FUNCTION

(* ---- K_TO_C.ST ---- *)
(*@PROPERTIES_EX@
TYPE: POU
LOCALE: 0
IEC_LANGUAGE: ST
PLC_TYPE: independent
PROC_TYPE: independent
GROUP: ENGINEERING.CONVERSION
*)
(*@KEY@:DESCRIPTION*)
version 1.1	19. aug 2009
programmer 	hugo
tested by	tobias

this function converts kelvin to celsius
(*@KEY@:END_DESCRIPTION*)
FUNCTION K_TO_C:REAL

(*Group:Default*)

VAR_INPUT
	KELVIN :	REAL;
END_VAR

(*@KEY@: WORKSHEET
NAME: K_TO_C
IEC_LANGUAGE: ST
*)
K_to_C := Kelvin + 273.15;

(* revision history

hm	4. aug 2006	rev 1.0
	original version

hm	19. aug 2009	rev 1.1
	fixed calculation error

*)

(*@KEY@: END_WORKSHEET *)
END_FUNCTION

(* ---- KMH_TO_MS.ST ---- *)
(*@PROPERTIES_EX@
TYPE: POU
LOCALE: 0
IEC_LANGUAGE: ST
PLC_TYPE: independent
PROC_TYPE: independent
GROUP: ENGINEERING.CONVERSION
*)
(*@KEY@:DESCRIPTION*)
version 1.1	6 jan 2007
programmer 	hugo
tested by	tobias

this function converts velocities from Kilometers / hour to Meters / Second
(*@KEY@:END_DESCRIPTION*)
FUNCTION KMH_TO_MS:REAL

(*Group:Default*)

VAR_INPUT
	KMH :	REAL;
END_VAR

(*@KEY@: WORKSHEET
NAME: KMH_TO_MS
IEC_LANGUAGE: ST
*)
KMH_TO_MS := kmh * 0.2777777777777;

(* revision history
hm	4. feb 2007		rev 1.0
	original version

hm	6. jan 2008		rev 1.1
	improved performance

*)
(*@KEY@: END_WORKSHEET *)
END_FUNCTION

(* ---- LANGEVIN.ST ---- *)
(*@PROPERTIES_EX@
TYPE: POU
LOCALE: 0
IEC_LANGUAGE: ST
PLC_TYPE: independent
PROC_TYPE: independent
GROUP: MATHEMATICAL.MATHE
*)
(*@KEY@:DESCRIPTION*)
version 1.2	10.mar. 2009
programmer 	hugo
tested by	tobias

this function calculates the langevin function
(*@KEY@:END_DESCRIPTION*)
FUNCTION LANGEVIN:REAL

(*Group:Default*)

VAR_INPUT
	X :	REAL;
END_VAR

(*@KEY@: WORKSHEET
NAME: LANGEVIN
IEC_LANGUAGE: ST
*)
IF X = 0.0 THEN
	LANGEVIN := 0.0;
ELSE
	LANGEVIN := COTH(X) - 1.0 / X;
END_IF;

(* revision history
hm	10.12.2007	rev 1.0
	original version

hm	11. mar 2008	rev 1.1
	changed formula to avoid problems when x = 0

hm	10. mar. 2009	rev 1.2
	real constants updated to new systax using dot

*)
(*@KEY@: END_WORKSHEET *)
END_FUNCTION

(* ---- LEAP_DAY.ST ---- *)
(*@PROPERTIES_EX@
TYPE: POU
LOCALE: 0
IEC_LANGUAGE: ST
PLC_TYPE: independent
PROC_TYPE: independent
GROUP: TIME_DATE
*)
(*@KEY@:DESCRIPTION*)
version 1.2	24. jan. 2011
programmer 	hugo
tested by	oscat

leap_day is true if the tested day is a leap day (29. of february).
(*@KEY@:END_DESCRIPTION*)
FUNCTION LEAP_DAY:BOOL

(*Group:Default*)

VAR_INPUT
	IDATE :	UDINT;
END_VAR

(*@KEY@: WORKSHEET
NAME: LEAP_DAY
IEC_LANGUAGE: ST
*)
LEAP_DAY := IDATE MOD UDINT#126230400 = UDINT#68169600;

(* change history

hm 	15. jun. 2008	rev 1.0
	original version

hm	7. oct. 2008	rev 1.1
	changed function month to month_of_date

hm	24. jan. 2011	rev 1.2
	improved performance
*)
(*@KEY@: END_WORKSHEET *)
END_FUNCTION

(* ---- LEAP_OF_DATE.ST ---- *)
(*@PROPERTIES_EX@
TYPE: POU
LOCALE: 0
IEC_LANGUAGE: ST
PLC_TYPE: independent
PROC_TYPE: independent
GROUP: TIME_DATE
*)
(*@KEY@:DESCRIPTION*)
version 1.3	28. jan. 2011
programmer 	hugo
tested by	tobias

leap_of_date is true if current year is a leap year
(*@KEY@:END_DESCRIPTION*)
FUNCTION LEAP_OF_DATE:BOOL

(*Group:Default*)

VAR_INPUT
	IDATE :	UDINT;
END_VAR

(*@KEY@: WORKSHEET
NAME: LEAP_OF_DATE
IEC_LANGUAGE: ST
*)
LEAP_OF_DATE := SHL(UDINT_TO_DWORD((idate + UDINT#43200) / UDINT#31557600), 30) = DWORD#16#80000000;

(* change history

2.10.2006		rev 1.1
the function now calls leap_year to accomodate further accuracy.
the function now works for any year from 1970 to 2100

8. jan 2008		rev 1.2
	improved code for better performance

28. jan. 2011	rev 1.3
	improved performance
*)
(*@KEY@: END_WORKSHEET *)
END_FUNCTION

(* ---- LEAP_YEAR.ST ---- *)
(*@PROPERTIES_EX@
TYPE: POU
LOCALE: 0
IEC_LANGUAGE: ST
PLC_TYPE: independent
PROC_TYPE: independent
GROUP: TIME_DATE
*)
(*@KEY@:DESCRIPTION*)
version 1.1	2 oct 2006
programmer 	hugo
tested by	tobias

leap_year is true if the tested year is a leap year
(*@KEY@:END_DESCRIPTION*)
FUNCTION LEAP_YEAR:BOOL

(*Group:Default*)

VAR_INPUT
	YEAR :	INT;
END_VAR

(*@KEY@: WORKSHEET
NAME: LEAP_YEAR
IEC_LANGUAGE: ST
*)
IF (year MOD INT#400) = INT#00 THEN
  leap_year := TRUE;
ELSIF (year MOD INT#100) = INT#00 THEN
  leap_year := FALSE;
ELSIF (year MOD INT#04) = INT#00 THEN
  leap_year := TRUE;
ELSE
  leap_year := FALSE;
END_IF;

(* change history

hm 	2.10.2006		rev 1.1
	the function now works for any year from 1970 up to 2100

hm	1. oct 2007		rev 1.2
	chaged code for higher performance
*)
(*@KEY@: END_WORKSHEET *)
END_FUNCTION

(* ---- LTIME_TO_UTC.ST ---- *)
(*@PROPERTIES_EX@
TYPE: POU
LOCALE: 0
IEC_LANGUAGE: ST
PLC_TYPE: independent
PROC_TYPE: independent
GROUP: TIME_DATE
*)
(*@KEY@:DESCRIPTION*)
version 1.7	13. nov. 2009
programmer 	hugo
tested by	oscat

LTIME_TO_UTC calculates UTC (World Time) from a local time LTIME. utc is calculated
by subtracting Time_Zone_Offset from ltime and if dst it true subtracting an additional hour from ltime.

(*@KEY@:END_DESCRIPTION*)
FUNCTION LTIME_TO_UTC:UDINT

(*Group:Default*)

VAR_INPUT
	LTIME :	UDINT;
	DST :	BOOL;
	TIME_ZONE_OFFSET :	INT;
END_VAR

(*@KEY@: WORKSHEET
NAME: LTIME_TO_UTC
IEC_LANGUAGE: ST
*)
LTIME_TO_UTC := LTIME - _INT_TO_UDINT(TIME_ZONE_OFFSET * 60);
IF DST THEN LTIME_TO_UTC := LTIME_TO_UTC - UDINT#3600; END_IF;

(* revision history
hm 5.7.2007		rev 1.0
	original version

hm 5.11.2007		rev 1.1
	replaced literal constant with variable because of error in möller ecp4 compiler

hm	12.nov 2007	rev 1.2
	changed Type of time_zone_offset from time to int to allow for time zones with negative offset

hm	8. dec 2007	rev 1.3
	corrected a problem with time_zone_offset

hm	14. oct. 2008	rev 1.4
	changed time_zone_offset from int to real to allow for half hour offset

hm	20. oct. 2006	rev 1.5
	changed time_zone_offset from Real to INT, now in Minutes

hm	27. feb. 2009	rev 1.6
	added type conversions to avoid warnings under codesys 3.0

ks	13. nov. 2009	rev 1.7
	corrected error in formula

*)
(*@KEY@: END_WORKSHEET *)
END_FUNCTION

(* ---- MANUAL.ST ---- *)
(*@PROPERTIES_EX@
TYPE: POU
LOCALE: 0
IEC_LANGUAGE: ST
PLC_TYPE: independent
PROC_TYPE: independent
GROUP: ENGINEERING.AUTOMATION
*)
(*@KEY@:DESCRIPTION*)
version 1.0	21. nov. 2008
programmer 	hugo
tested by	oscat

MANUAL is a manual override for digital signals.
when on and off = FALSE, the output follows IN.
ON = TRUE forces the output high, and OFF = TRUE forces the output low.
(*@KEY@:END_DESCRIPTION*)
FUNCTION MANUAL:BOOL

(*Group:Default*)

VAR_INPUT
	IN :	BOOL;
	ON :	BOOL;
	OFF :	BOOL;
END_VAR

(*@KEY@: WORKSHEET
NAME: MANUAL
IEC_LANGUAGE: ST
*)
MANUAL := NOT OFF AND (IN OR ON);

(* revision history
hm	21. nov 2008	rev 1.0
	original version

*)
(*@KEY@: END_WORKSHEET *)
END_FUNCTION

(* ---- MAX3.ST ---- *)
(*@PROPERTIES_EX@
TYPE: POU
LOCALE: 0
IEC_LANGUAGE: ST
PLC_TYPE: independent
PROC_TYPE: independent
GROUP: MATHEMATICAL.MATHE
*)
(*@KEY@:DESCRIPTION*)
version 1.1	18. mar. 2011
programmer 	hugo
tested by	tobias

this function returns the highest of 3 real values
(*@KEY@:END_DESCRIPTION*)
FUNCTION MAX3:REAL

(*Group:Default*)

VAR_INPUT
	IN1 :	REAL;
	IN2 :	REAL;
	IN3 :	REAL;
END_VAR

(*@KEY@: WORKSHEET
NAME: MAX3
IEC_LANGUAGE: ST
*)
MAX3 := MAX(MAX(IN1,IN2),IN3);

(* revision history
hm	1.1.2007	rev 1.0
	original release

hm	18. mar. 2011	rev 1.1
	improve performance

*)
(*@KEY@: END_WORKSHEET *)
END_FUNCTION

(* ---- MID3.ST ---- *)
(*@PROPERTIES_EX@
TYPE: POU
LOCALE: 0
IEC_LANGUAGE: ST
PLC_TYPE: independent
PROC_TYPE: independent
GROUP: MATHEMATICAL.MATHE
*)
(*@KEY@:DESCRIPTION*)
version 1.2	18. mar. 2011
programmer 	hugo
tested by	tobias

returns the mid value of 3 real inputs.
(*@KEY@:END_DESCRIPTION*)
FUNCTION MID3:REAL

(*Group:Default*)

VAR_INPUT
	IN1 :	REAL;
	IN2 :	REAL;
	IN3 :	REAL;
END_VAR

VAR
	_IN1 :	REAL;
	_IN2 :	REAL;
	_IN3 :	REAL;
END_VAR

(*@KEY@: WORKSHEET
NAME: MID3
IEC_LANGUAGE: ST
*)
_IN1 := IN1; (* VAR_INPUT auf Variablen umkopieren , da diese schreibgeschützt sind *)
_IN2 := IN2;
_IN3 := IN3;

IF _IN1 > _IN2 THEN MID3 := _IN1; _IN1 := _IN2; _IN2 := MID3; END_IF;
IF _IN2 > _IN3 THEN _IN2 := _IN3; END_IF;
MID3 := SEL(_IN1 > _IN2, _IN2, _IN1);

(*
hm	1.1.2007	rev 1.1
	rewrote the function for better performance

hm	18. mar. 2011	rev 1.2
	improve performance
*)
(*@KEY@: END_WORKSHEET *)
END_FUNCTION

(* ---- MIN3.ST ---- *)
(*@PROPERTIES_EX@
TYPE: POU
LOCALE: 0
IEC_LANGUAGE: ST
PLC_TYPE: independent
PROC_TYPE: independent
GROUP: MATHEMATICAL.MATHE
*)
(*@KEY@:DESCRIPTION*)
version 1.1	18. mar. 2011
programmer 	hugo
tested by	tobias

this function returns the lowest of 3 real values
(*@KEY@:END_DESCRIPTION*)
FUNCTION MIN3:REAL

(*Group:Default*)

VAR_INPUT
	IN1 :	REAL;
	IN2 :	REAL;
	IN3 :	REAL;
END_VAR

(*@KEY@: WORKSHEET
NAME: MIN3
IEC_LANGUAGE: ST
*)
MIN3 := MIN(MIN(IN1,IN2),IN3);

(* revision history
hm	1.1.2007	rev 1.0
	original release

hm	18. mar. 2011	rev 1.1
	improve performance

*)
(*@KEY@: END_WORKSHEET *)
END_FUNCTION

(* ---- MINUTE.ST ---- *)
(*@PROPERTIES_EX@
TYPE: POU
LOCALE: 0
IEC_LANGUAGE: ST
PLC_TYPE: independent
PROC_TYPE: independent
GROUP: TIME_DATE
*)
(*@KEY@:DESCRIPTION*)
version 1.1	2 oct 2006
programmer 	hugo
tested by	tobias

extracts the minutes out of TOD truncating the ceconds
(*@KEY@:END_DESCRIPTION*)
FUNCTION MINUTE:INT

(*Group:Default*)

VAR_INPUT
	ITOD :	UDINT;
END_VAR

(*@KEY@: WORKSHEET
NAME: MINUTE
IEC_LANGUAGE: ST
*)
minute := UDINT_TO_INT((itod / UDINT#60000) - ((itod / UDINT#3600000) * UDINT#60));

(* change history

2.10.2006 changes name of input to itod

*)
(*@KEY@: END_WORKSHEET *)
END_FUNCTION

(* ---- MINUTE_OF_DT.ST ---- *)
(*@PROPERTIES_EX@
TYPE: POU
LOCALE: 0
IEC_LANGUAGE: ST
PLC_TYPE: independent
PROC_TYPE: independent
GROUP: TIME_DATE
*)
(*@KEY@:DESCRIPTION*)
version 1.0	6. jun. 2008
programmer 	oscat
tested BY	oscat

MINUTE_OF_DT returns the current minute (minute of the hour) of a DT variable
(*@KEY@:END_DESCRIPTION*)
FUNCTION MINUTE_OF_DT:INT

(*Group:Default*)

VAR_INPUT
	XDT :	UDINT;
END_VAR

(*@KEY@: WORKSHEET
NAME: MINUTE_OF_DT
IEC_LANGUAGE: ST
*)
MINUTE_OF_DT := UDINT_TO_INT((XDT MOD UDINT#3600) / UDINT#60);

(* revision history
hm		6.9.2008	rev 1.0
	original version

*)
(*@KEY@: END_WORKSHEET *)
END_FUNCTION

(* ---- MINUTE_TO_TIME.ST ---- *)
(*@PROPERTIES_EX@
TYPE: POU
LOCALE: 0
IEC_LANGUAGE: ST
PLC_TYPE: independent
PROC_TYPE: independent
GROUP: TIME_DATE
*)
(*@KEY@:DESCRIPTION*)
version 1.2	24. feb. 2009
programmer 	hugo
tested by	oscat

converts an amount of minutes in real to time
(*@KEY@:END_DESCRIPTION*)
FUNCTION MINUTE_TO_TIME:TIME

(*Group:Default*)

VAR_INPUT
	IN :	REAL;
END_VAR

(*@KEY@: WORKSHEET
NAME: MINUTE_TO_TIME
IEC_LANGUAGE: ST
*)
minute_to_time := UDINT_TO_TIME(_REAL_TO_UDINT(IN * 60000.0));

(* revision history
hm		4. aug 2006	rev 1.0
	original version

hm		14. mar 2008	rev 1.1
	rounded the input after the last digit

*)
(*@KEY@: END_WORKSHEET *)
END_FUNCTION

(* ---- MIX.ST ---- *)
(*@PROPERTIES_EX@
TYPE: POU
LOCALE: 0
IEC_LANGUAGE: ST
PLC_TYPE: independent
PROC_TYPE: independent
GROUP: ENGINEERING.SIGNAL_PROCESSING
*)
(*@KEY@:DESCRIPTION*)
version 1.1	10. mar. 2009
programmer 	hugo
tested by	tobias

MIX is an analog Mixer. The Output is (1-M)*A + M*B.

(*@KEY@:END_DESCRIPTION*)
FUNCTION MIX:REAL

(*Group:Default*)

VAR_INPUT
	A :	REAL;
	B :	REAL;
	M :	REAL;
END_VAR

(*@KEY@: WORKSHEET
NAME: MIX
IEC_LANGUAGE: ST
*)
MIX := (1.0 - M) * A + M * B;

(* revision history
hm	19. Nov 2007	rev 1.0
	original version

hm	10. mar 2009	rev 1.1
	real constants updated to new systax using dot

*)
(*@KEY@: END_WORKSHEET *)
END_FUNCTION

(* ---- MODR.ST ---- *)
(*@PROPERTIES_EX@
TYPE: POU
LOCALE: 0
IEC_LANGUAGE: ST
PLC_TYPE: independent
PROC_TYPE: independent
GROUP: MATHEMATICAL.MATHE
*)
(*@KEY@:DESCRIPTION*)
version 1.5	10. mar. 2009
programmer 	hugo
tested by	tobias

this is a modulo funtion for real numbers
modr(5.5,2.5) = 0.5

(*@KEY@:END_DESCRIPTION*)
FUNCTION MODR:REAL

(*Group:Default*)

VAR_INPUT
	IN :	REAL;
	DIVI :	REAL;
END_VAR

(*@KEY@: WORKSHEET
NAME: MODR
IEC_LANGUAGE: ST
*)
IF divi = 0.0 THEN
	MODR := 0.0;
ELSE
	MODR := in - DINT_TO_REAL(FLOOR2(in / divi)) * divi;
END_IF;

(* revision history

hm	4. aug.2006		rev 1.0

hm	28. jan.2007	rev 1.1
	modr(x,0) will deliver the result 0

hm	21. mar 2008	rev 1.2
	use D_trunc for compatibility reasons

hm	4. apr. 2008	rev 1.3
	added type conversion to avoid warnings under codesys 3.0

hm	31. oct. 2008	rev 1.4
	changed algorithm to the more common version using floor instead of TRUNC

hm	10. mar. 2009	rev 1.5
	real constants updated to new systax using dot

*)
(*@KEY@: END_WORKSHEET *)
END_FUNCTION

(* ---- MONTH_BEGIN.ST ---- *)
(*@PROPERTIES_EX@
TYPE: POU
LOCALE: 0
IEC_LANGUAGE: ST
PLC_TYPE: independent
PROC_TYPE: independent
GROUP: TIME_DATE
*)
(*@KEY@:DESCRIPTION*)
version 1.0	15. jun. 2008
programmer 	hugo
tested by	oscat

returns the date for the first day of the current month in the current year.
(*@KEY@:END_DESCRIPTION*)
FUNCTION MONTH_BEGIN:UDINT

(*Group:Default*)

VAR_INPUT
	IDATE :	UDINT;
END_VAR

(*@KEY@: WORKSHEET
NAME: MONTH_BEGIN
IEC_LANGUAGE: ST
*)
MONTH_BEGIN := idate - _INT_TO_UDINT(DAY_OF_MONTH(idate) - 1) * UDINT#86400;

(* revision history
hm	15. JUN: 2008	rev 1.0
	original version

*)
(*@KEY@: END_WORKSHEET *)
END_FUNCTION

(* ---- MONTH_END.ST ---- *)
(*@PROPERTIES_EX@
TYPE: POU
LOCALE: 0
IEC_LANGUAGE: ST
PLC_TYPE: independent
PROC_TYPE: independent
GROUP: TIME_DATE
*)
(*@KEY@:DESCRIPTION*)
version 1.1	7. oct. 2008
programmer 	hugo
tested by	oscat

returns the date for the last day of the current month in the current year.
(*@KEY@:END_DESCRIPTION*)
FUNCTION MONTH_END:UDINT

(*Group:Default*)

VAR_INPUT
	IDATE :	UDINT;
END_VAR

(*@KEY@: WORKSHEET
NAME: MONTH_END
IEC_LANGUAGE: ST
*)
MONTH_END := SET_DATE(YEAR_OF_DATE(idate),MONTH_OF_DATE(idate)+1,1) - UDINT#86400;

(* revision history
hm	15. jun. 2008	rev 1.0
	original version

hm	7. oct. 2008	rev 1.1
	changed function year to year_of_date
	changed function month to month_of_date

*)
(*@KEY@: END_WORKSHEET *)
END_FUNCTION

(* ---- MONTH_OF_DATE.ST ---- *)
(*@PROPERTIES_EX@
TYPE: POU
LOCALE: 0
IEC_LANGUAGE: ST
PLC_TYPE: independent
PROC_TYPE: independent
GROUP: TIME_DATE
*)
(*@KEY@:DESCRIPTION*)
version 1.3	27. mar. 2009
programmer 	hugo
tested by	tobias

returns the current month of the year.
(*@KEY@:END_DESCRIPTION*)
FUNCTION MONTH_OF_DATE:INT

(*Group:Default*)

VAR_INPUT
	IDATE :	UDINT;
END_VAR

(*@KEY@: WORKSHEET
NAME: MONTH_OF_DATE
IEC_LANGUAGE: ST
*)
MONTH_OF_DATE := DAY_OF_YEAR(idate);
IF MONTH_OF_DATE < 32 THEN
	MONTH_OF_DATE := 1;
ELSIF LEAP_OF_DATE(IDATE) THEN
	MONTH_OF_DATE := (MONTH_OF_DATE * 53 + 1668) / 1623;
ELSE
	MONTH_OF_DATE := (MONTH_OF_DATE * 53 + 1700) / 1620;
END_IF;

(* code for rev 1.2
MONTH_OF_DATE := DAY_OF_YEAR(IDATE);
IF LEAP_OF_DATE(IDATE) THEN
	CASE MONTH_OF_DATE OF
		1..31 	:	MONTH_OF_DATE := 1;
		32..60	:	MONTH_OF_DATE := 2;
		61..91	:	MONTH_OF_DATE := 3;
		92..121 :	MONTH_OF_DATE := 4;
		122..152:	MONTH_OF_DATE := 5;
		153..182:	MONTH_OF_DATE := 6;
		183..213:	MONTH_OF_DATE := 7;
		214..244:	MONTH_OF_DATE := 8;
		245..274:	MONTH_OF_DATE := 9;
		275..305:	MONTH_OF_DATE := 10;
		306..335:	MONTH_OF_DATE := 11;
		336..366:	MONTH_OF_DATE := 12;
	END_CASE;
ELSE
	CASE MONTH_OF_DATE OF
		1..31 	:	MONTH_OF_DATE := 1;
		32..59	:	MONTH_OF_DATE := 2;
		60..90	:	MONTH_OF_DATE := 3;
		91..120 :	MONTH_OF_DATE := 4;
		121..151:	MONTH_OF_DATE := 5;
		152..181:	MONTH_OF_DATE := 6;
		182..212:	MONTH_OF_DATE := 7;
		213..243:	MONTH_OF_DATE := 8;
		244..273:	MONTH_OF_DATE := 9;
		274..304:	MONTH_OF_DATE := 10;
		305..334:	MONTH_OF_DATE := 11;
		335..365:	MONTH_OF_DATE := 12;
	END_CASE;
END_IF;
*)

(* revision history
hm	1. aug 2006	rev 1.0
	original version

hm	1. okt 2007	rev 1.1
	replaced old code (string conversion) with mathematics
	the execution time is now multiple times faster.

hm	7. oct. 2008	rev 1.2
	changed name of function from month to MONTH_OF_DATE

hm	27. mar. 2009	rev 1.3
	new improved code

*)
(*@KEY@: END_WORKSHEET *)
END_FUNCTION

(* ---- MS_TO_BFT.ST ---- *)
(*@PROPERTIES_EX@
TYPE: POU
LOCALE: 0
IEC_LANGUAGE: ST
PLC_TYPE: independent
PROC_TYPE: independent
GROUP: ENGINEERING.CONVERSION
*)
(*@KEY@:DESCRIPTION*)
version 1.0	12. jun 2008
programmer 	hugo
tested by	oscdat

this function converts wind speed from M/s to beaufort
(*@KEY@:END_DESCRIPTION*)
FUNCTION MS_TO_BFT:INT

(*Group:Default*)

VAR_INPUT
	MS :	REAL;
END_VAR

(*@KEY@: WORKSHEET
NAME: MS_TO_BFT
IEC_LANGUAGE: ST
*)
MS_TO_BFT := REAL_TO_INT(EXPT(MS * 1.196172, 0.666667));

(* revision history
hm	12. 6. 2008		rev 1.0
	original version

*)
(*@KEY@: END_WORKSHEET *)
END_FUNCTION
